KUKA KRL program: f1_Kuka_APT212T02S12.SRC

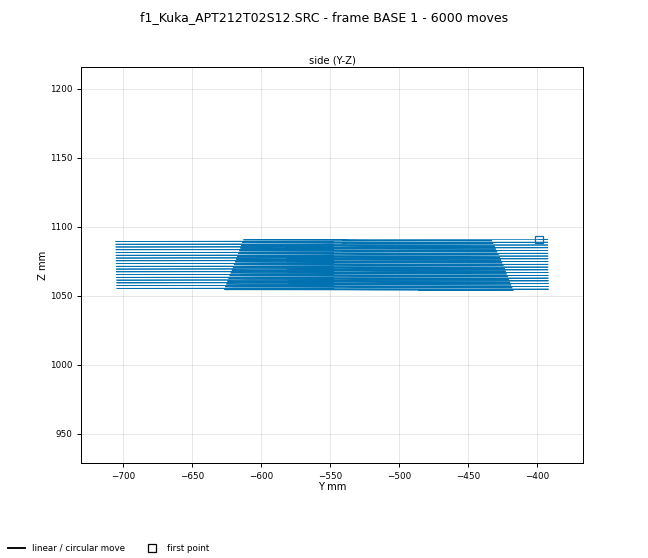
[picture p0: tool path of f1_Kuka_APT212T02S12.SRC in frame BASE 1, 6000 of 6001 moves have a stored position in this frame; points joined in program order, loops and branches not executed]
&ACCESS RVP
&REL 2
&PARAM TEMPLATE = C:\KRC\Roboter\Template\vorgabe
&PARAM EDITMASK = *
DEF f1_Kuka_APT212T02S12()


;FOLD INI;%{PE}%V3.2.0,%MKUKATPBASIS,%CINIT,%VCOMMON,%P
  ;FOLD BAS INI;%{E}%V3.2.0,%MKUKATPBASIS,%CINIT,%VINIT,%P
    GLOBAL INTERRUPT DECL 3 WHEN $STOPMESS==TRUE DO IR_STOPM ( )
    INTERRUPT ON 3
    BAS (#INITMOV,0 )
  ;ENDFOLD (BAS INI)
  ;FOLD USER INI;%{E}%V3.2.0,%MKUKATPUSER,%CINIT,%VINIT,%P
    ;Make your modifications here
  ;ENDFOLD (USER INI)
;ENDFOLD (INI)


;*** Make Null PTP Move
  PTP $pos_act

;*** Auto Load The Correct TOOL Data
  $tool=tool_data[2]

;*** Auto Load The Correct BASE Data
  $base=base_data[1]

  $ADVANCE = 5

;*** Restate Last Velocity
MMPM(30000.0)
SetRPM(8000)
LIN {X -0.086,Y -398.427,Z 1090.884,A 0.000,B 0.000,C 90.000,E1 15.190} C_DIS
LIN {X -0.036,Y -396.041,Z 1090.882,A 0.000,B 0.000,C 90.000,E1 14.773} C_DIS
LIN {X 0.107,Y -394.257,Z 1090.880,A 0.000,B 0.000,C 90.000,E1 14.356} C_DIS
LIN {X 0.038,Y -393.540,Z 1090.879,A 0.000,B 0.000,C 90.000,E1 14.189} C_DIS
LIN {X 0.038,Y -392.338,Z 1090.876,A 0.000,B 0.000,C 90.000,E1 13.647} C_DIS
LIN {X 0.042,Y -392.056,Z 1090.872,A 0.000,B 0.000,C 90.000,E1 12.939} C_DIS
LIN {X -0.016,Y -392.577,Z 1090.868,A 0.000,B 0.000,C 90.000,E1 12.243} C_DIS
LIN {X -0.109,Y -394.607,Z 1090.860,A 0.000,B 0.000,C 90.000,E1 10.838} C_DIS
LIN {X 0.062,Y -400.114,Z 1090.844,A 0.000,B 0.000,C 90.000,E1 7.992} C_DIS
LIN {X -0.050,Y -404.941,Z 1090.833,A 0.000,B 0.000,C 90.000,E1 5.910} C_DIS
LIN {X -0.108,Y -406.949,Z 1090.828,A 0.000,B 0.000,C 90.000,E1 5.049} C_DIS
LIN {X -0.130,Y -409.374,Z 1090.824,A 0.000,B 0.000,C 90.000,E1 4.359} C_DIS
LIN {X 0.208,Y -412.372,Z 1090.821,A 0.000,B 0.000,C 90.000,E1 3.784} C_DIS
LIN {X -0.071,Y -415.342,Z 1090.819,A 0.000,B 0.000,C 90.000,E1 3.498} C_DIS
LIN {X 0.069,Y -416.809,Z 1090.819,A 0.000,B 0.000,C 90.000,E1 3.326} C_DIS
LIN {X -0.093,Y -424.402,Z 1090.816,A 0.000,B 0.000,C 90.000,E1 2.808} C_DIS
LIN {X 0.127,Y -432.552,Z 1090.813,A 0.000,B 0.000,C 90.000,E1 2.236} C_DIS
LIN {X -0.175,Y -448.840,Z 1090.807,A 0.000,B 0.000,C 90.000,E1 1.203} C_DIS
LIN {X 0.179,Y -470.911,Z 1090.799,A 0.000,B 0.000,C 90.000,E1 359.771} C_DIS
LIN {X -0.123,Y -480.615,Z 1090.796,A 0.000,B 0.000,C 90.000,E1 359.198} C_DIS
LIN {X -0.067,Y -490.234,Z 1090.792,A 0.000,B 0.000,C 90.000,E1 358.568} C_DIS
LIN {X -0.141,Y -501.141,Z 1090.788,A 0.000,B 0.000,C 90.000,E1 357.822} C_DIS
LIN {X -0.002,Y -508.747,Z 1090.785,A 0.000,B 0.000,C 90.000,E1 357.249} C_DIS
LIN {X -0.176,Y -517.486,Z 1090.781,A 0.000,B 0.000,C 90.000,E1 356.560} C_DIS
LIN {X 0.062,Y -523.142,Z 1090.778,A 0.000,B 0.000,C 90.000,E1 356.045} C_DIS
LIN {X 0.124,Y -528.481,Z 1090.775,A 0.000,B 0.000,C 90.000,E1 355.527} C_DIS
LIN {X -0.033,Y -533.756,Z 1090.772,A 0.000,B 0.000,C 90.000,E1 355.008} C_DIS
LIN {X -0.006,Y -539.738,Z 1090.768,A 0.000,B 0.000,C 90.000,E1 354.318} C_DIS
LIN {X -0.098,Y -545.312,Z 1090.765,A 0.000,B 0.000,C 90.000,E1 353.628} C_DIS
LIN {X 0.005,Y -549.510,Z 1090.761,A 0.000,B 0.000,C 90.000,E1 353.053} C_DIS
LIN {X -0.044,Y -554.087,Z 1090.758,A 0.000,B 0.000,C 90.000,E1 352.356} C_DIS
LIN {X 0.122,Y -557.472,Z 1090.755,A 0.000,B 0.000,C 90.000,E1 351.781} C_DIS
LIN {X 0.146,Y -561.205,Z 1090.751,A 0.000,B 0.000,C 90.000,E1 351.084} C_DIS
LIN {X 0.207,Y -564.647,Z 1090.747,A 0.000,B 0.000,C 90.000,E1 350.387} C_DIS
LIN {X -0.087,Y -568.925,Z 1090.741,A 0.000,B 0.000,C 90.000,E1 349.454} C_DIS
LIN {X 0.100,Y -573.356,Z 1090.735,A 0.000,B 0.000,C 90.000,E1 348.342} C_DIS
LIN {X -0.002,Y -578.374,Z 1090.728,A 0.000,B 0.000,C 90.000,E1 346.992} C_DIS
LIN {X 0.202,Y -583.916,Z 1090.719,A 0.000,B 0.000,C 90.000,E1 345.353} C_DIS
LIN {X 0.003,Y -588.183,Z 1090.711,A 0.000,B 0.000,C 90.000,E1 344.031} C_DIS
LIN {X 0.030,Y -591.458,Z 1090.705,A 0.000,B 0.000,C 90.000,E1 342.960} C_DIS
LIN {X -0.029,Y -595.407,Z 1090.698,A 0.000,B 0.000,C 90.000,E1 341.638} C_DIS
LIN {X -0.187,Y -597.634,Z 1090.694,A 0.000,B 0.000,C 90.000,E1 340.859} C_DIS
LIN {X 0.046,Y -600.855,Z 1090.686,A 0.000,B 0.000,C 90.000,E1 339.518} C_DIS
LIN {X 0.066,Y -603.171,Z 1090.680,A 0.000,B 0.000,C 90.000,E1 338.465} C_DIS
LIN {X 0.124,Y -605.226,Z 1090.675,A 0.000,B 0.000,C 90.000,E1 337.411} C_DIS
LIN {X 0.209,Y -607.002,Z 1090.669,A 0.000,B 0.000,C 90.000,E1 336.357} C_DIS
LIN {X -0.245,Y -608.528,Z 1090.663,A 0.000,B 0.000,C 90.000,E1 335.357} C_DIS
LIN {X 0.127,Y -609.836,Z 1090.657,A 0.000,B 0.000,C 90.000,E1 334.280} C_DIS
LIN {X -0.030,Y -610.932,Z 1090.651,A 0.000,B 0.000,C 90.000,E1 333.256} C_DIS
LIN {X -0.211,Y -611.924,Z 1090.644,A 0.000,B 0.000,C 90.000,E1 331.975} C_DIS
LIN {X -0.023,Y -612.377,Z 1090.640,A 0.000,B 0.000,C 90.000,E1 331.179} C_DIS
LIN {X 0.141,Y -612.615,Z 1090.634,A 0.000,B 0.000,C 90.000,E1 330.127} C_DIS
LIN {X 0.342,Y -612.436,Z 1090.630,A 0.000,B 0.000,C 90.000,E1 329.331} C_DIS
LIN {X 0.017,Y -612.074,Z 1090.625,A 0.000,B 0.000,C 90.000,E1 328.584} C_DIS
LIN {X 0.210,Y -611.462,Z 1090.621,A 0.000,B 0.000,C 90.000,E1 327.788} C_DIS
LIN {X 0.156,Y -610.184,Z 1090.615,A 0.000,B 0.000,C 90.000,E1 326.755} C_DIS
LIN {X 0.088,Y -608.451,Z 1090.610,A 0.000,B 0.000,C 90.000,E1 325.722} C_DIS
LIN {X 0.262,Y -606.198,Z 1090.602,A 0.000,B 0.000,C 90.000,E1 324.402} C_DIS
LIN {X -0.099,Y -604.017,Z 1090.595,A 0.000,B 0.000,C 90.000,E1 323.130} C_DIS
LIN {X -0.134,Y -601.862,Z 1090.588,A 0.000,B 0.000,C 90.000,E1 321.823} C_DIS
LIN {X 0.148,Y -600.611,Z 1090.583,A 0.000,B 0.000,C 90.000,E1 321.009} C_DIS
LIN {X -0.208,Y -599.661,Z 1090.581,A 0.000,B 0.000,C 90.000,E1 320.517} C_DIS
LIN {X 0.031,Y -599.310,Z 1090.579,A 0.000,B 0.000,C 90.000,E1 320.231} C_DIS
LIN {X -0.190,Y -598.777,Z 1090.578,A 0.000,B 0.000,C 90.000,E1 319.989} C_DIS
LIN {X -0.177,Y -598.069,Z 1090.575,A 0.000,B 0.000,C 90.000,E1 319.461} C_DIS
LIN {X -0.169,Y -597.234,Z 1090.572,A 0.000,B 0.000,C 90.000,E1 318.933} C_DIS
LIN {X -0.168,Y -596.422,Z 1090.569,A 0.000,B 0.000,C 90.000,E1 318.405} C_DIS
LIN {X 0.214,Y -594.488,Z 1090.563,A 0.000,B 0.000,C 90.000,E1 317.310} C_DIS
LIN {X -0.269,Y -592.283,Z 1090.557,A 0.000,B 0.000,C 90.000,E1 316.296} C_DIS
LIN {X -0.134,Y -590.462,Z 1090.553,A 0.000,B 0.000,C 90.000,E1 315.486} C_DIS
LIN {X -0.170,Y -586.110,Z 1090.542,A 0.000,B 0.000,C 90.000,E1 313.623} C_DIS
LIN {X 0.151,Y -584.801,Z 1090.539,A 0.000,B 0.000,C 90.000,E1 313.056} C_DIS
LIN {X -0.129,Y -580.589,Z 1090.530,A 0.000,B 0.000,C 90.000,E1 311.472} C_DIS
LIN {X 0.142,Y -579.157,Z 1090.527,A 0.000,B 0.000,C 90.000,E1 310.906} C_DIS
LIN {X 0.176,Y -576.205,Z 1090.523,A 0.000,B 0.000,C 90.000,E1 310.092} C_DIS
LIN {X 0.037,Y -574.143,Z 1090.520,A 0.000,B 0.000,C 90.000,E1 309.564} C_DIS
LIN {X 0.155,Y -569.404,Z 1090.514,A 0.000,B 0.000,C 90.000,E1 308.463} C_DIS
LIN {X -0.031,Y -564.794,Z 1090.509,A 0.000,B 0.000,C 90.000,E1 307.523} C_DIS
LIN {X 0.190,Y -561.998,Z 1090.505,A 0.000,B 0.000,C 90.000,E1 306.950} C_DIS
LIN {X -0.178,Y -558.216,Z 1090.502,A 0.000,B 0.000,C 90.000,E1 306.297} C_DIS
LIN {X -0.008,Y -554.762,Z 1090.499,A 0.000,B 0.000,C 90.000,E1 305.724} C_DIS
LIN {X -0.057,Y -551.848,Z 1090.496,A 0.000,B 0.000,C 90.000,E1 305.311} C_DIS
LIN {X -0.064,Y -547.711,Z 1090.492,A 0.000,B 0.000,C 90.000,E1 304.612} C_DIS
LIN {X -0.016,Y -545.861,Z 1090.491,A 0.000,B 0.000,C 90.000,E1 304.326} C_DIS
LIN {X -0.244,Y -542.889,Z 1090.488,A 0.000,B 0.000,C 90.000,E1 303.785} C_DIS
LIN {X 0.261,Y -540.814,Z 1090.484,A 0.000,B 0.000,C 90.000,E1 303.166} C_DIS
LIN {X 0.155,Y -539.184,Z 1090.480,A 0.000,B 0.000,C 90.000,E1 302.467} C_DIS
LIN {X 0.179,Y -538.819,Z 1090.479,A 0.000,B 0.000,C 90.000,E1 302.133} C_DIS
LIN {X -0.101,Y -538.609,Z 1090.477,A 0.000,B 0.000,C 90.000,E1 301.878} C_DIS
LIN {X -0.096,Y -538.156,Z 1090.475,A 0.000,B 0.000,C 90.000,E1 301.592} C_DIS
LIN {X 0.085,Y -537.926,Z 1090.474,A 0.000,B 0.000,C 90.000,E1 301.288} C_DIS
LIN {X 0.150,Y -537.874,Z 1090.472,A 0.000,B 0.000,C 90.000,E1 301.003} C_DIS
LIN {X 0.147,Y -537.993,Z 1090.471,A 0.000,B 0.000,C 90.000,E1 300.718} C_DIS
LIN {X -0.132,Y -537.654,Z 1090.469,A 0.000,B 0.000,C 90.000,E1 300.463} C_DIS
LIN {X -0.308,Y -538.599,Z 1090.447,A 0.000,B 0.000,C 90.000,E1 296.488} C_DIS
LIN {X 0.034,Y -539.190,Z 1090.439,A 0.000,B 0.000,C 90.000,E1 295.027} C_DIS
LIN {X 0.166,Y -539.672,Z 1090.431,A 0.000,B 0.000,C 90.000,E1 293.590} C_DIS
LIN {X 0.033,Y -540.215,Z 1090.422,A 0.000,B 0.000,C 90.000,E1 291.897} C_DIS
LIN {X -0.030,Y -540.561,Z 1090.414,A 0.000,B 0.000,C 90.000,E1 290.482} C_DIS
LIN {X -0.275,Y -540.656,Z 1090.406,A 0.000,B 0.000,C 90.000,E1 289.087} C_DIS
LIN {X -0.227,Y -540.529,Z 1090.400,A 0.000,B 0.000,C 90.000,E1 287.946} C_DIS
LIN {X 0.039,Y -540.294,Z 1090.392,A 0.000,B 0.000,C 90.000,E1 286.496} C_DIS
LIN {X 0.203,Y -539.799,Z 1090.382,A 0.000,B 0.000,C 90.000,E1 284.773} C_DIS
LIN {X 0.153,Y -539.168,Z 1090.374,A 0.000,B 0.000,C 90.000,E1 283.355} C_DIS
LIN {X -0.027,Y -538.495,Z 1090.366,A 0.000,B 0.000,C 90.000,E1 281.951} C_DIS
LIN {X -0.218,Y -537.760,Z 1090.359,A 0.000,B 0.000,C 90.000,E1 280.546} C_DIS
LIN {X 0.010,Y -537.088,Z 1090.351,A 0.000,B 0.000,C 90.000,E1 279.095} C_DIS
LIN {X -0.268,Y -536.057,Z 1090.339,A 0.000,B 0.000,C 90.000,E1 277.125} C_DIS
LIN {X -0.103,Y -535.245,Z 1090.330,A 0.000,B 0.000,C 90.000,E1 275.391} C_DIS
LIN {X -0.045,Y -534.093,Z 1090.317,A 0.000,B 0.000,C 90.000,E1 273.094} C_DIS
LIN {X -0.069,Y -533.037,Z 1090.304,A 0.000,B 0.000,C 90.000,E1 270.802} C_DIS
LIN {X -0.101,Y -532.288,Z 1090.297,A 0.000,B 0.000,C 90.000,E1 269.370} C_DIS
LIN {X -0.147,Y -531.316,Z 1090.287,A 0.000,B 0.000,C 90.000,E1 267.650} C_DIS
LIN {X -0.200,Y -530.464,Z 1090.279,A 0.000,B 0.000,C 90.000,E1 266.216} C_DIS
LIN {X -0.238,Y -529.531,Z 1090.271,A 0.000,B 0.000,C 90.000,E1 264.780} C_DIS
LIN {X -0.226,Y -528.880,Z 1090.266,A 0.000,B 0.000,C 90.000,E1 263.913} C_DIS
LIN {X -0.279,Y -528.109,Z 1090.261,A 0.000,B 0.000,C 90.000,E1 263.053} C_DIS
LIN {X -0.216,Y -526.239,Z 1090.252,A 0.000,B 0.000,C 90.000,E1 261.310} C_DIS
LIN {X -0.164,Y -524.132,Z 1090.240,A 0.000,B 0.000,C 90.000,E1 259.275} C_DIS
LIN {X -0.103,Y -522.944,Z 1090.234,A 0.000,B 0.000,C 90.000,E1 258.105} C_DIS
LIN {X -0.056,Y -521.283,Z 1090.224,A 0.000,B 0.000,C 90.000,E1 256.353} C_DIS
LIN {X 0.190,Y -519.569,Z 1090.214,A 0.000,B 0.000,C 90.000,E1 254.574} C_DIS
LIN {X 0.023,Y -517.402,Z 1090.203,A 0.000,B 0.000,C 90.000,E1 252.543} C_DIS
LIN {X -0.050,Y -515.164,Z 1090.192,A 0.000,B 0.000,C 90.000,E1 250.496} C_DIS
LIN {X -0.208,Y -513.874,Z 1090.185,A 0.000,B 0.000,C 90.000,E1 249.337} C_DIS
LIN {X -0.076,Y -512.072,Z 1090.177,A 0.000,B 0.000,C 90.000,E1 247.847} C_DIS
LIN {X 0.027,Y -510.158,Z 1090.169,A 0.000,B 0.000,C 90.000,E1 246.357} C_DIS
LIN {X -0.016,Y -508.348,Z 1090.162,A 0.000,B 0.000,C 90.000,E1 245.177} C_DIS
LIN {X -0.023,Y -505.922,Z 1090.154,A 0.000,B 0.000,C 90.000,E1 243.691} C_DIS
LIN {X 0.004,Y -504.492,Z 1090.149,A 0.000,B 0.000,C 90.000,E1 242.794} C_DIS
LIN {X -0.062,Y -502.029,Z 1090.141,A 0.000,B 0.000,C 90.000,E1 241.307} C_DIS
LIN {X 0.101,Y -498.891,Z 1090.131,A 0.000,B 0.000,C 90.000,E1 239.488} C_DIS
LIN {X 0.130,Y -496.801,Z 1090.124,A 0.000,B 0.000,C 90.000,E1 238.280} C_DIS
LIN {X 0.122,Y -495.153,Z 1090.119,A 0.000,B 0.000,C 90.000,E1 237.375} C_DIS
LIN {X -0.205,Y -491.745,Z 1090.109,A 0.000,B 0.000,C 90.000,E1 235.595} C_DIS
LIN {X -0.177,Y -488.784,Z 1090.100,A 0.000,B 0.000,C 90.000,E1 234.069} C_DIS
LIN {X -0.146,Y -486.406,Z 1090.094,A 0.000,B 0.000,C 90.000,E1 232.844} C_DIS
LIN {X -0.025,Y -483.277,Z 1090.085,A 0.000,B 0.000,C 90.000,E1 231.295} C_DIS
LIN {X -0.080,Y -480.708,Z 1090.078,A 0.000,B 0.000,C 90.000,E1 230.070} C_DIS
LIN {X -0.329,Y -476.867,Z 1090.068,A 0.000,B 0.000,C 90.000,E1 228.243} C_DIS
LIN {X -0.151,Y -472.084,Z 1090.054,A 0.000,B 0.000,C 90.000,E1 225.729} C_DIS
LIN {X -0.208,Y -468.066,Z 1090.042,A 0.000,B 0.000,C 90.000,E1 223.542} C_DIS
LIN {X 0.172,Y -465.067,Z 1090.033,A 0.000,B 0.000,C 90.000,E1 221.919} C_DIS
LIN {X 0.233,Y -461.505,Z 1090.022,A 0.000,B 0.000,C 90.000,E1 220.011} C_DIS
LIN {X -0.115,Y -458.564,Z 1090.014,A 0.000,B 0.000,C 90.000,E1 218.463} C_DIS
LIN {X 0.208,Y -455.116,Z 1090.003,A 0.000,B 0.000,C 90.000,E1 216.503} C_DIS
LIN {X 0.195,Y -452.321,Z 1089.994,A 0.000,B 0.000,C 90.000,E1 214.898} C_DIS
LIN {X 0.046,Y -450.006,Z 1089.987,A 0.000,B 0.000,C 90.000,E1 213.627} C_DIS
LIN {X -0.015,Y -447.787,Z 1089.980,A 0.000,B 0.000,C 90.000,E1 212.339} C_DIS
LIN {X 0.019,Y -444.410,Z 1089.969,A 0.000,B 0.000,C 90.000,E1 210.384} C_DIS
LIN {X -0.036,Y -440.736,Z 1089.956,A 0.000,B 0.000,C 90.000,E1 208.103} C_DIS
LIN {X 0.101,Y -435.648,Z 1089.936,A 0.000,B 0.000,C 90.000,E1 204.463} C_DIS
LIN {X 0.037,Y -433.167,Z 1089.923,A 0.000,B 0.000,C 90.000,E1 202.153} C_DIS
LIN {X -0.118,Y -432.631,Z 1089.916,A 0.000,B 0.000,C 90.000,E1 200.844} C_DIS
LIN {X 0.148,Y -432.819,Z 1089.910,A 0.000,B 0.000,C 90.000,E1 199.812} C_DIS
LIN {X 0.191,Y -433.420,Z 1089.906,A 0.000,B 0.000,C 90.000,E1 199.141} C_DIS
LIN {X -0.081,Y -435.004,Z 1089.901,A 0.000,B 0.000,C 90.000,E1 198.181} C_DIS
LIN {X -0.025,Y -436.647,Z 1089.897,A 0.000,B 0.000,C 90.000,E1 197.511} C_DIS
LIN {X 0.159,Y -439.745,Z 1089.892,A 0.000,B 0.000,C 90.000,E1 196.496} C_DIS
LIN {X 0.112,Y -444.855,Z 1089.885,A 0.000,B 0.000,C 90.000,E1 195.190} C_DIS
LIN {X 0.164,Y -456.278,Z 1089.870,A 0.000,B 0.000,C 90.000,E1 192.591} C_DIS
LIN {X -0.058,Y -460.863,Z 1089.865,A 0.000,B 0.000,C 90.000,E1 191.658} C_DIS
LIN {X -0.140,Y -465.504,Z 1089.859,A 0.000,B 0.000,C 90.000,E1 190.715} C_DIS
LIN {X -0.075,Y -468.813,Z 1089.856,A 0.000,B 0.000,C 90.000,E1 190.074} C_DIS
LIN {X -0.194,Y -472.599,Z 1089.852,A 0.000,B 0.000,C 90.000,E1 189.321} C_DIS
LIN {X 0.098,Y -474.289,Z 1089.850,A 0.000,B 0.000,C 90.000,E1 188.973} C_DIS
LIN {X -0.103,Y -479.620,Z 1089.844,A 0.000,B 0.000,C 90.000,E1 187.936} C_DIS
LIN {X 0.069,Y -485.064,Z 1089.838,A 0.000,B 0.000,C 90.000,E1 186.834} C_DIS
LIN {X -0.236,Y -490.322,Z 1089.832,A 0.000,B 0.000,C 90.000,E1 185.796} C_DIS
LIN {X -0.134,Y -496.944,Z 1089.824,A 0.000,B 0.000,C 90.000,E1 184.416} C_DIS
LIN {X -0.233,Y -504.229,Z 1089.816,A 0.000,B 0.000,C 90.000,E1 182.922} C_DIS
LIN {X 0.197,Y -512.902,Z 1089.806,A 0.000,B 0.000,C 90.000,E1 181.088} C_DIS
LIN {X -0.155,Y -520.097,Z 1089.798,A 0.000,B 0.000,C 90.000,E1 179.656} C_DIS
LIN {X 0.156,Y -527.331,Z 1089.790,A 0.000,B 0.000,C 90.000,E1 178.165} C_DIS
LIN {X -0.198,Y -536.562,Z 1089.780,A 0.000,B 0.000,C 90.000,E1 176.331} C_DIS
LIN {X -0.084,Y -543.539,Z 1089.772,A 0.000,B 0.000,C 90.000,E1 174.894} C_DIS
LIN {X 0.255,Y -551.899,Z 1089.762,A 0.000,B 0.000,C 90.000,E1 173.166} C_DIS
LIN {X -0.260,Y -560.082,Z 1089.753,A 0.000,B 0.000,C 90.000,E1 171.546} C_DIS
LIN {X -0.131,Y -566.707,Z 1089.745,A 0.000,B 0.000,C 90.000,E1 170.151} C_DIS
LIN {X 0.114,Y -573.062,Z 1089.738,A 0.000,B 0.000,C 90.000,E1 168.757} C_DIS
LIN {X 0.254,Y -578.637,Z 1089.731,A 0.000,B 0.000,C 90.000,E1 167.521} C_DIS
LIN {X 0.119,Y -582.785,Z 1089.726,A 0.000,B 0.000,C 90.000,E1 166.589} C_DIS
LIN {X -0.254,Y -588.499,Z 1089.718,A 0.000,B 0.000,C 90.000,E1 165.283} C_DIS
LIN {X -0.221,Y -592.795,Z 1089.712,A 0.000,B 0.000,C 90.000,E1 164.212} C_DIS
LIN {X -0.129,Y -596.808,Z 1089.706,A 0.000,B 0.000,C 90.000,E1 163.142} C_DIS
LIN {X 0.194,Y -600.573,Z 1089.700,A 0.000,B 0.000,C 90.000,E1 162.054} C_DIS
LIN {X 0.295,Y -604.968,Z 1089.693,A 0.000,B 0.000,C 90.000,E1 160.732} C_DIS
LIN {X 0.098,Y -609.053,Z 1089.686,A 0.000,B 0.000,C 90.000,E1 159.444} C_DIS
LIN {X 0.014,Y -612.200,Z 1089.680,A 0.000,B 0.000,C 90.000,E1 158.411} C_DIS
LIN {X 0.229,Y -614.406,Z 1089.676,A 0.000,B 0.000,C 90.000,E1 157.614} C_DIS
LIN {X -0.169,Y -618.738,Z 1089.667,A 0.000,B 0.000,C 90.000,E1 156.102} C_DIS
LIN {X 0.096,Y -621.386,Z 1089.661,A 0.000,B 0.000,C 90.000,E1 155.049} C_DIS
LIN {X 0.097,Y -624.653,Z 1089.654,A 0.000,B 0.000,C 90.000,E1 153.768} C_DIS
LIN {X 0.141,Y -627.168,Z 1089.649,A 0.000,B 0.000,C 90.000,E1 152.743} C_DIS
LIN {X -0.293,Y -630.738,Z 1089.640,A 0.000,B 0.000,C 90.000,E1 151.257} C_DIS
LIN {X 0.157,Y -633.517,Z 1089.633,A 0.000,B 0.000,C 90.000,E1 149.950} C_DIS
LIN {X -0.074,Y -636.759,Z 1089.625,A 0.000,B 0.000,C 90.000,E1 148.456} C_DIS
LIN {X 0.306,Y -639.862,Z 1089.616,A 0.000,B 0.000,C 90.000,E1 146.914} C_DIS
LIN {X 0.155,Y -642.295,Z 1089.609,A 0.000,B 0.000,C 90.000,E1 145.674} C_DIS
LIN {X -0.072,Y -645.172,Z 1089.601,A 0.000,B 0.000,C 90.000,E1 144.196} C_DIS
LIN {X 0.145,Y -647.954,Z 1089.593,A 0.000,B 0.000,C 90.000,E1 142.683} C_DIS
LIN {X 0.419,Y -650.745,Z 1089.584,A 0.000,B 0.000,C 90.000,E1 141.170} C_DIS
LIN {X -0.270,Y -653.698,Z 1089.576,A 0.000,B 0.000,C 90.000,E1 139.747} C_DIS
LIN {X -0.054,Y -657.592,Z 1089.565,A 0.000,B 0.000,C 90.000,E1 137.757} C_DIS
LIN {X -0.206,Y -661.174,Z 1089.556,A 0.000,B 0.000,C 90.000,E1 136.053} C_DIS
LIN {X -0.310,Y -666.280,Z 1089.544,A 0.000,B 0.000,C 90.000,E1 133.866} C_DIS
LIN {X 0.183,Y -669.940,Z 1089.536,A 0.000,B 0.000,C 90.000,E1 132.366} C_DIS
LIN {X -0.117,Y -674.850,Z 1089.525,A 0.000,B 0.000,C 90.000,E1 130.458} C_DIS
LIN {X -0.209,Y -679.639,Z 1089.514,A 0.000,B 0.000,C 90.000,E1 128.543} C_DIS
LIN {X 0.175,Y -683.417,Z 1089.506,A 0.000,B 0.000,C 90.000,E1 127.076} C_DIS
LIN {X 0.186,Y -686.458,Z 1089.500,A 0.000,B 0.000,C 90.000,E1 125.884} C_DIS
LIN {X 0.054,Y -688.731,Z 1089.494,A 0.000,B 0.000,C 90.000,E1 124.945} C_DIS
LIN {X 0.358,Y -692.196,Z 1089.486,A 0.000,B 0.000,C 90.000,E1 123.499} C_DIS
LIN {X 0.123,Y -695.084,Z 1089.480,A 0.000,B 0.000,C 90.000,E1 122.339} C_DIS
LIN {X -0.075,Y -697.857,Z 1089.473,A 0.000,B 0.000,C 90.000,E1 121.180} C_DIS
LIN {X 0.089,Y -699.296,Z 1089.469,A 0.000,B 0.000,C 90.000,E1 120.463} C_DIS
LIN {X -0.067,Y -700.996,Z 1089.464,A 0.000,B 0.000,C 90.000,E1 119.539} C_DIS
LIN {X 0.136,Y -701.989,Z 1089.460,A 0.000,B 0.000,C 90.000,E1 118.821} C_DIS
LIN {X 0.350,Y -702.820,Z 1089.456,A 0.000,B 0.000,C 90.000,E1 118.103} C_DIS
LIN {X 0.192,Y -703.825,Z 1089.450,A 0.000,B 0.000,C 90.000,E1 116.950} C_DIS
LIN {X -0.296,Y -705.017,Z 1089.442,A 0.000,B 0.000,C 90.000,E1 115.591} C_DIS
LIN {X 0.279,Y -705.272,Z 1089.439,A 0.000,B 0.000,C 90.000,E1 115.079} C_DIS
LIN {X -0.081,Y -705.294,Z 1089.437,A 0.000,B 0.000,C 90.000,E1 114.643} C_DIS
LIN {X 0.204,Y -704.753,Z 1089.434,A 0.000,B 0.000,C 90.000,E1 114.155} C_DIS
LIN {X -0.153,Y -704.352,Z 1089.433,A 0.000,B 0.000,C 90.000,E1 113.951} C_DIS
LIN {X 0.132,Y -702.683,Z 1089.430,A 0.000,B 0.000,C 90.000,E1 113.462} C_DIS
LIN {X -0.234,Y -701.490,Z 1089.429,A 0.000,B 0.000,C 90.000,E1 113.259} C_DIS
LIN {X 0.033,Y -697.713,Z 1089.427,A 0.000,B 0.000,C 90.000,E1 112.770} C_DIS
LIN {X 0.163,Y -696.456,Z 1089.426,A 0.000,B 0.000,C 90.000,E1 112.642} C_DIS
LIN {X 0.291,Y -694.466,Z 1089.425,A 0.000,B 0.000,C 90.000,E1 112.514} C_DIS
LIN {X 0.169,Y -687.151,Z 1089.423,A 0.000,B 0.000,C 90.000,E1 112.206} C_DIS
LIN {X -0.051,Y -684.897,Z 1089.423,A 0.000,B 0.000,C 90.000,E1 112.153} C_DIS
LIN {X 0.024,Y -675.825,Z 1089.422,A 0.000,B 0.000,C 90.000,E1 112.025} C_DIS
LIN {X -0.028,Y -604.808,Z 1089.422,A 0.000,B 0.000,C 90.000,E1 112.025} C_DIS
LIN {X -0.164,Y -600.949,Z 1089.421,A 0.000,B 0.000,C 90.000,E1 111.844} C_DIS
LIN {X -0.082,Y -596.421,Z 1089.420,A 0.000,B 0.000,C 90.000,E1 111.535} C_DIS
LIN {X 0.109,Y -586.219,Z 1089.415,A 0.000,B 0.000,C 90.000,E1 110.684} C_DIS
LIN {X -0.207,Y -576.459,Z 1089.410,A 0.000,B 0.000,C 90.000,E1 109.885} C_DIS
LIN {X -0.103,Y -575.095,Z 1089.410,A 0.000,B 0.000,C 90.000,E1 109.758} C_DIS
LIN {X -0.227,Y -569.062,Z 1089.407,A 0.000,B 0.000,C 90.000,E1 109.322} C_DIS
LIN {X 0.087,Y -560.876,Z 1089.404,A 0.000,B 0.000,C 90.000,E1 108.779} C_DIS
LIN {X -0.023,Y -554.397,Z 1089.402,A 0.000,B 0.000,C 90.000,E1 108.417} C_DIS
LIN {X 0.181,Y -549.521,Z 1089.401,A 0.000,B 0.000,C 90.000,E1 108.055} C_DIS
LIN {X 0.056,Y -548.089,Z 1089.399,A 0.000,B 0.000,C 90.000,E1 107.873} C_DIS
LIN {X 0.013,Y -548.062,Z 1089.399,A 0.000,B 0.000,C 90.000,E1 107.873} C_DIS
LIN {X -0.276,Y -547.700,Z 1089.398,A 0.000,B 0.000,C 90.000,E1 107.583} C_DIS
LIN {X -0.075,Y -547.929,Z 1089.394,A 0.000,B 0.000,C 90.000,E1 106.858} C_DIS
LIN {X -0.169,Y -548.528,Z 1089.389,A 0.000,B 0.000,C 90.000,E1 106.024} C_DIS
LIN {X -0.239,Y -549.880,Z 1089.378,A 0.000,B 0.000,C 90.000,E1 104.064} C_DIS
LIN {X 0.122,Y -551.468,Z 1089.367,A 0.000,B 0.000,C 90.000,E1 102.063} C_DIS
LIN {X 0.166,Y -552.809,Z 1089.359,A 0.000,B 0.000,C 90.000,E1 100.658} C_DIS
LIN {X -0.254,Y -554.877,Z 1089.349,A 0.000,B 0.000,C 90.000,E1 98.746} C_DIS
LIN {X -0.253,Y -556.387,Z 1089.341,A 0.000,B 0.000,C 90.000,E1 97.352} C_DIS
LIN {X 0.122,Y -557.648,Z 1089.335,A 0.000,B 0.000,C 90.000,E1 96.201} C_DIS
LIN {X -0.036,Y -558.705,Z 1089.328,A 0.000,B 0.000,C 90.000,E1 95.106} C_DIS
LIN {X 0.247,Y -559.426,Z 1089.324,A 0.000,B 0.000,C 90.000,E1 94.245} C_DIS
LIN {X 0.190,Y -560.344,Z 1089.316,A 0.000,B 0.000,C 90.000,E1 92.865} C_DIS
LIN {X 0.019,Y -560.983,Z 1089.310,A 0.000,B 0.000,C 90.000,E1 91.776} C_DIS
LIN {X 0.037,Y -561.803,Z 1089.301,A 0.000,B 0.000,C 90.000,E1 90.115} C_DIS
LIN {X 0.074,Y -562.503,Z 1089.292,A 0.000,B 0.000,C 90.000,E1 88.453} C_DIS
LIN {X 0.033,Y -563.084,Z 1089.284,A 0.000,B 0.000,C 90.000,E1 87.078} C_DIS
LIN {X 0.038,Y -563.621,Z 1089.276,A 0.000,B 0.000,C 90.000,E1 85.698} C_DIS
LIN {X 0.058,Y -564.161,Z 1089.269,A 0.000,B 0.000,C 90.000,E1 84.318} C_DIS
LIN {X -0.166,Y -564.757,Z 1089.258,A 0.000,B 0.000,C 90.000,E1 82.413} C_DIS
LIN {X -0.072,Y -565.248,Z 1089.250,A 0.000,B 0.000,C 90.000,E1 81.027} C_DIS
LIN {X -0.106,Y -566.034,Z 1089.240,A 0.000,B 0.000,C 90.000,E1 79.106} C_DIS
LIN {X -0.179,Y -566.772,Z 1089.230,A 0.000,B 0.000,C 90.000,E1 77.465} C_DIS
LIN {X 0.242,Y -567.996,Z 1089.218,A 0.000,B 0.000,C 90.000,E1 75.227} C_DIS
LIN {X 0.073,Y -569.712,Z 1089.204,A 0.000,B 0.000,C 90.000,E1 72.779} C_DIS
LIN {X -0.017,Y -571.020,Z 1089.195,A 0.000,B 0.000,C 90.000,E1 71.148} C_DIS
LIN {X -0.086,Y -572.452,Z 1089.186,A 0.000,B 0.000,C 90.000,E1 69.518} C_DIS
LIN {X -0.283,Y -573.181,Z 1089.182,A 0.000,B 0.000,C 90.000,E1 68.720} C_DIS
LIN {X -0.070,Y -574.770,Z 1089.171,A 0.000,B 0.000,C 90.000,E1 66.794} C_DIS
LIN {X 0.199,Y -575.835,Z 1089.164,A 0.000,B 0.000,C 90.000,E1 65.409} C_DIS
LIN {X -0.182,Y -576.961,Z 1089.155,A 0.000,B 0.000,C 90.000,E1 63.819} C_DIS
LIN {X 0.231,Y -577.998,Z 1089.146,A 0.000,B 0.000,C 90.000,E1 62.153} C_DIS
LIN {X -0.216,Y -578.818,Z 1089.138,A 0.000,B 0.000,C 90.000,E1 60.845} C_DIS
LIN {X 0.139,Y -579.590,Z 1089.130,A 0.000,B 0.000,C 90.000,E1 59.459} C_DIS
LIN {X -0.144,Y -580.458,Z 1089.121,A 0.000,B 0.000,C 90.000,E1 57.867} C_DIS
LIN {X -0.126,Y -580.980,Z 1089.115,A 0.000,B 0.000,C 90.000,E1 56.786} C_DIS
LIN {X -0.090,Y -581.617,Z 1089.108,A 0.000,B 0.000,C 90.000,E1 55.435} C_DIS
LIN {X -0.188,Y -582.250,Z 1089.099,A 0.000,B 0.000,C 90.000,E1 53.829} C_DIS
LIN {X -0.005,Y -582.501,Z 1089.094,A 0.000,B 0.000,C 90.000,E1 53.004} C_DIS
LIN {X 0.240,Y -582.741,Z 1089.089,A 0.000,B 0.000,C 90.000,E1 51.904} C_DIS
LIN {X 0.021,Y -582.694,Z 1089.080,A 0.000,B 0.000,C 90.000,E1 50.312} C_DIS
LIN {X 0.198,Y -582.443,Z 1089.074,A 0.000,B 0.000,C 90.000,E1 49.218} C_DIS
LIN {X 0.267,Y -582.187,Z 1089.069,A 0.000,B 0.000,C 90.000,E1 48.405} C_DIS
LIN {X -0.085,Y -581.522,Z 1089.060,A 0.000,B 0.000,C 90.000,E1 46.824} C_DIS
LIN {X 0.089,Y -580.962,Z 1089.054,A 0.000,B 0.000,C 90.000,E1 45.729} C_DIS
LIN {X -0.163,Y -580.147,Z 1089.048,A 0.000,B 0.000,C 90.000,E1 44.676} C_DIS
LIN {X -0.155,Y -579.400,Z 1089.044,A 0.000,B 0.000,C 90.000,E1 43.866} C_DIS
LIN {X -0.012,Y -578.194,Z 1089.038,A 0.000,B 0.000,C 90.000,E1 42.771} C_DIS
LIN {X 0.111,Y -576.737,Z 1089.032,A 0.000,B 0.000,C 90.000,E1 41.676} C_DIS
LIN {X 0.120,Y -575.463,Z 1089.027,A 0.000,B 0.000,C 90.000,E1 40.862} C_DIS
LIN {X -0.174,Y -573.643,Z 1089.021,A 0.000,B 0.000,C 90.000,E1 39.806} C_DIS
LIN {X -0.360,Y -570.873,Z 1089.014,A 0.000,B 0.000,C 90.000,E1 38.463} C_DIS
LIN {X 0.041,Y -568.929,Z 1089.009,A 0.000,B 0.000,C 90.000,E1 37.604} C_DIS
LIN {X -0.033,Y -566.684,Z 1089.004,A 0.000,B 0.000,C 90.000,E1 36.790} C_DIS
LIN {X -0.015,Y -564.120,Z 1089.000,A 0.000,B 0.000,C 90.000,E1 35.964} C_DIS
LIN {X 0.098,Y -563.221,Z 1088.998,A 0.000,B 0.000,C 90.000,E1 35.678} C_DIS
LIN {X -0.276,Y -559.027,Z 1088.992,A 0.000,B 0.000,C 90.000,E1 34.612} C_DIS
LIN {X -0.328,Y -555.516,Z 1088.988,A 0.000,B 0.000,C 90.000,E1 33.785} C_DIS
LIN {X 0.042,Y -551.533,Z 1088.983,A 0.000,B 0.000,C 90.000,E1 32.911} C_DIS
LIN {X 0.069,Y -546.568,Z 1088.977,A 0.000,B 0.000,C 90.000,E1 31.926} C_DIS
LIN {X 0.198,Y -541.282,Z 1088.972,A 0.000,B 0.000,C 90.000,E1 30.924} C_DIS
LIN {X 0.117,Y -534.473,Z 1088.966,A 0.000,B 0.000,C 90.000,E1 29.795} C_DIS
LIN {X 0.124,Y -529.787,Z 1088.962,A 0.000,B 0.000,C 90.000,E1 29.077} C_DIS
LIN {X 0.243,Y -525.777,Z 1088.958,A 0.000,B 0.000,C 90.000,E1 28.487} C_DIS
LIN {X -0.217,Y -522.681,Z 1088.956,A 0.000,B 0.000,C 90.000,E1 28.103} C_DIS
LIN {X 0.049,Y -514.540,Z 1088.950,A 0.000,B 0.000,C 90.000,E1 27.052} C_DIS
LIN {X 0.141,Y -508.048,Z 1088.946,A 0.000,B 0.000,C 90.000,E1 26.309} C_DIS
LIN {X 0.231,Y -502.730,Z 1088.943,A 0.000,B 0.000,C 90.000,E1 25.720} C_DIS
LIN {X -0.019,Y -494.568,Z 1088.938,A 0.000,B 0.000,C 90.000,E1 24.899} C_DIS
LIN {X -0.042,Y -488.960,Z 1088.935,A 0.000,B 0.000,C 90.000,E1 24.335} C_DIS
LIN {X -0.107,Y -477.381,Z 1088.929,A 0.000,B 0.000,C 90.000,E1 23.259} C_DIS
LIN {X -0.054,Y -471.540,Z 1088.926,A 0.000,B 0.000,C 90.000,E1 22.717} C_DIS
LIN {X 0.000,Y -457.967,Z 1088.920,A 0.000,B 0.000,C 90.000,E1 21.535} C_DIS
LIN {X -0.172,Y -441.851,Z 1088.912,A 0.000,B 0.000,C 90.000,E1 20.120} C_DIS
LIN {X -0.132,Y -430.227,Z 1088.906,A 0.000,B 0.000,C 90.000,E1 19.014} C_DIS
LIN {X 0.092,Y -416.281,Z 1088.897,A 0.000,B 0.000,C 90.000,E1 17.511} C_DIS
LIN {X -0.045,Y -405.620,Z 1088.890,A 0.000,B 0.000,C 90.000,E1 16.260} C_DIS
LIN {X 0.133,Y -399.045,Z 1088.885,A 0.000,B 0.000,C 90.000,E1 15.371} C_DIS
LIN {X -0.048,Y -395.343,Z 1088.882,A 0.000,B 0.000,C 90.000,E1 14.773} C_DIS
LIN {X 0.131,Y -393.924,Z 1088.880,A 0.000,B 0.000,C 90.000,E1 14.356} C_DIS
LIN {X 0.061,Y -393.206,Z 1088.879,A 0.000,B 0.000,C 90.000,E1 14.189} C_DIS
LIN {X -0.091,Y -392.129,Z 1088.875,A 0.000,B 0.000,C 90.000,E1 13.592} C_DIS
LIN {X 0.057,Y -392.164,Z 1088.871,A 0.000,B 0.000,C 90.000,E1 12.771} C_DIS
LIN {X 0.064,Y -393.130,Z 1088.866,A 0.000,B 0.000,C 90.000,E1 11.883} C_DIS
LIN {X -0.156,Y -397.974,Z 1088.850,A 0.000,B 0.000,C 90.000,E1 9.086} C_DIS
LIN {X 0.004,Y -404.983,Z 1088.833,A 0.000,B 0.000,C 90.000,E1 5.910} C_DIS
LIN {X -0.038,Y -406.506,Z 1088.829,A 0.000,B 0.000,C 90.000,E1 5.220} C_DIS
LIN {X -0.070,Y -407.479,Z 1088.827,A 0.000,B 0.000,C 90.000,E1 4.878} C_DIS
LIN {X -0.078,Y -409.273,Z 1088.824,A 0.000,B 0.000,C 90.000,E1 4.359} C_DIS
LIN {X -0.166,Y -412.135,Z 1088.821,A 0.000,B 0.000,C 90.000,E1 3.841} C_DIS
LIN {X 0.037,Y -412.697,Z 1088.821,A 0.000,B 0.000,C 90.000,E1 3.726} C_DIS
LIN {X -0.051,Y -417.157,Z 1088.818,A 0.000,B 0.000,C 90.000,E1 3.269} C_DIS
LIN {X -0.126,Y -421.852,Z 1088.816,A 0.000,B 0.000,C 90.000,E1 2.922} C_DIS
LIN {X 0.056,Y -429.349,Z 1088.813,A 0.000,B 0.000,C 90.000,E1 2.407} C_DIS
LIN {X -0.176,Y -448.932,Z 1088.806,A 0.000,B 0.000,C 90.000,E1 1.146} C_DIS
LIN {X 0.000,Y -466.750,Z 1088.800,A 0.000,B 0.000,C 90.000,E1 360.000} C_DIS
LIN {X -0.227,Y -478.221,Z 1088.796,A 0.000,B 0.000,C 90.000,E1 359.312} C_DIS
LIN {X -0.180,Y -486.222,Z 1088.793,A 0.000,B 0.000,C 90.000,E1 358.797} C_DIS
LIN {X 0.154,Y -492.517,Z 1088.791,A 0.000,B 0.000,C 90.000,E1 358.339} C_DIS
LIN {X 0.031,Y -503.476,Z 1088.787,A 0.000,B 0.000,C 90.000,E1 357.593} C_DIS
LIN {X 0.092,Y -509.565,Z 1088.784,A 0.000,B 0.000,C 90.000,E1 357.135} C_DIS
LIN {X -0.066,Y -516.942,Z 1088.781,A 0.000,B 0.000,C 90.000,E1 356.560} C_DIS
LIN {X 0.174,Y -523.948,Z 1088.777,A 0.000,B 0.000,C 90.000,E1 355.927} C_DIS
LIN {X -0.222,Y -527.993,Z 1088.775,A 0.000,B 0.000,C 90.000,E1 355.584} C_DIS
LIN {X 0.168,Y -533.306,Z 1088.772,A 0.000,B 0.000,C 90.000,E1 355.008} C_DIS
LIN {X 0.275,Y -539.325,Z 1088.769,A 0.000,B 0.000,C 90.000,E1 354.318} C_DIS
LIN {X 0.178,Y -544.973,Z 1088.765,A 0.000,B 0.000,C 90.000,E1 353.628} C_DIS
LIN {X -0.108,Y -549.141,Z 1088.762,A 0.000,B 0.000,C 90.000,E1 353.109} C_DIS
LIN {X -0.160,Y -553.773,Z 1088.758,A 0.000,B 0.000,C 90.000,E1 352.413} C_DIS
LIN {X 0.004,Y -557.227,Z 1088.755,A 0.000,B 0.000,C 90.000,E1 351.837} C_DIS
LIN {X 0.027,Y -561.014,Z 1088.751,A 0.000,B 0.000,C 90.000,E1 351.141} C_DIS
LIN {X 0.086,Y -564.506,Z 1088.747,A 0.000,B 0.000,C 90.000,E1 350.443} C_DIS
LIN {X 0.175,Y -567.644,Z 1088.743,A 0.000,B 0.000,C 90.000,E1 349.746} C_DIS
LIN {X 0.156,Y -571.162,Z 1088.739,A 0.000,B 0.000,C 90.000,E1 348.926} C_DIS
LIN {X 0.057,Y -574.391,Z 1088.734,A 0.000,B 0.000,C 90.000,E1 348.117} C_DIS
LIN {X -0.251,Y -578.431,Z 1088.728,A 0.000,B 0.000,C 90.000,E1 347.061} C_DIS
LIN {X 0.088,Y -584.048,Z 1088.719,A 0.000,B 0.000,C 90.000,E1 345.408} C_DIS
LIN {X 0.138,Y -589.193,Z 1088.710,A 0.000,B 0.000,C 90.000,E1 343.795} C_DIS
LIN {X 0.178,Y -592.460,Z 1088.704,A 0.000,B 0.000,C 90.000,E1 342.725} C_DIS
LIN {X -0.127,Y -595.647,Z 1088.698,A 0.000,B 0.000,C 90.000,E1 341.692} C_DIS
LIN {X 0.181,Y -598.589,Z 1088.692,A 0.000,B 0.000,C 90.000,E1 340.604} C_DIS
LIN {X -0.124,Y -601.774,Z 1088.685,A 0.000,B 0.000,C 90.000,E1 339.316} C_DIS
LIN {X -0.305,Y -604.052,Z 1088.679,A 0.000,B 0.000,C 90.000,E1 338.284} C_DIS
LIN {X -0.239,Y -606.102,Z 1088.673,A 0.000,B 0.000,C 90.000,E1 337.230} C_DIS
LIN {X -0.198,Y -608.248,Z 1088.666,A 0.000,B 0.000,C 90.000,E1 335.921} C_DIS
LIN {X 0.172,Y -609.679,Z 1088.660,A 0.000,B 0.000,C 90.000,E1 334.845} C_DIS
LIN {X -0.021,Y -611.223,Z 1088.653,A 0.000,B 0.000,C 90.000,E1 333.563} C_DIS
LIN {X -0.157,Y -612.119,Z 1088.647,A 0.000,B 0.000,C 90.000,E1 332.538} C_DIS
LIN {X -0.286,Y -612.890,Z 1088.642,A 0.000,B 0.000,C 90.000,E1 331.513} C_DIS
LIN {X -0.085,Y -613.194,Z 1088.637,A 0.000,B 0.000,C 90.000,E1 330.717} C_DIS
LIN {X 0.123,Y -613.371,Z 1088.633,A 0.000,B 0.000,C 90.000,E1 329.921} C_DIS
LIN {X 0.020,Y -613.189,Z 1088.629,A 0.000,B 0.000,C 90.000,E1 329.154} C_DIS
LIN {X -0.022,Y -612.670,Z 1088.623,A 0.000,B 0.000,C 90.000,E1 328.122} C_DIS
LIN {X 0.173,Y -611.851,Z 1088.619,A 0.000,B 0.000,C 90.000,E1 327.327} C_DIS
LIN {X -0.161,Y -610.954,Z 1088.614,A 0.000,B 0.000,C 90.000,E1 326.580} C_DIS
LIN {X -0.163,Y -609.783,Z 1088.610,A 0.000,B 0.000,C 90.000,E1 325.801} C_DIS
LIN {X -0.243,Y -608.114,Z 1088.604,A 0.000,B 0.000,C 90.000,E1 324.769} C_DIS
LIN {X -0.307,Y -605.653,Z 1088.595,A 0.000,B 0.000,C 90.000,E1 323.210} C_DIS
LIN {X -0.015,Y -602.496,Z 1088.584,A 0.000,B 0.000,C 90.000,E1 321.090} C_DIS
LIN {X -0.062,Y -599.891,Z 1088.574,A 0.000,B 0.000,C 90.000,E1 319.256} C_DIS
LIN {X 0.366,Y -598.362,Z 1088.568,A 0.000,B 0.000,C 90.000,E1 318.162} C_DIS
LIN {X -0.065,Y -596.606,Z 1088.562,A 0.000,B 0.000,C 90.000,E1 317.148} C_DIS
LIN {X 0.321,Y -594.642,Z 1088.556,A 0.000,B 0.000,C 90.000,E1 316.053} C_DIS
LIN {X 0.063,Y -592.969,Z 1088.552,A 0.000,B 0.000,C 90.000,E1 315.283} C_DIS
LIN {X -0.213,Y -591.337,Z 1088.547,A 0.000,B 0.000,C 90.000,E1 314.514} C_DIS
LIN {X 0.151,Y -590.312,Z 1088.544,A 0.000,B 0.000,C 90.000,E1 313.947} C_DIS
LIN {X -0.051,Y -586.879,Z 1088.535,A 0.000,B 0.000,C 90.000,E1 312.366} C_DIS
LIN {X 0.061,Y -585.196,Z 1088.531,A 0.000,B 0.000,C 90.000,E1 311.553} C_DIS
LIN {X 0.279,Y -582.693,Z 1088.525,A 0.000,B 0.000,C 90.000,E1 310.458} C_DIS
LIN {X 0.009,Y -581.982,Z 1088.523,A 0.000,B 0.000,C 90.000,E1 310.216} C_DIS
LIN {X 0.237,Y -578.366,Z 1088.517,A 0.000,B 0.000,C 90.000,E1 309.116} C_DIS
LIN {X 0.061,Y -574.101,Z 1088.511,A 0.000,B 0.000,C 90.000,E1 308.051} C_DIS
LIN {X 0.182,Y -569.480,Z 1088.505,A 0.000,B 0.000,C 90.000,E1 306.950} C_DIS
LIN {X -0.015,Y -567.030,Z 1088.502,A 0.000,B 0.000,C 90.000,E1 306.423} C_DIS
LIN {X 0.104,Y -561.186,Z 1088.496,A 0.000,B 0.000,C 90.000,E1 305.311} C_DIS
LIN {X 0.178,Y -556.779,Z 1088.492,A 0.000,B 0.000,C 90.000,E1 304.612} C_DIS
LIN {X 0.141,Y -554.043,Z 1088.490,A 0.000,B 0.000,C 90.000,E1 304.199} C_DIS
LIN {X 0.023,Y -547.768,Z 1088.485,A 0.000,B 0.000,C 90.000,E1 303.372} C_DIS
LIN {X -0.104,Y -546.814,Z 1088.485,A 0.000,B 0.000,C 90.000,E1 303.245} C_DIS
LIN {X 0.067,Y -546.099,Z 1088.484,A 0.000,B 0.000,C 90.000,E1 303.086} C_DIS
LIN {X -0.190,Y -544.341,Z 1088.482,A 0.000,B 0.000,C 90.000,E1 302.832} C_DIS
LIN {X -0.033,Y -542.110,Z 1088.479,A 0.000,B 0.000,C 90.000,E1 302.260} C_DIS
LIN {X -0.299,Y -541.189,Z 1088.478,A 0.000,B 0.000,C 90.000,E1 302.005} C_DIS
LIN {X 0.042,Y -540.146,Z 1088.475,A 0.000,B 0.000,C 90.000,E1 301.544} C_DIS
LIN {X -0.085,Y -539.478,Z 1088.473,A 0.000,B 0.000,C 90.000,E1 301.131} C_DIS
LIN {X 0.332,Y -539.599,Z 1088.472,A 0.000,B 0.000,C 90.000,E1 300.924} C_DIS
LIN {X 0.058,Y -539.304,Z 1088.470,A 0.000,B 0.000,C 90.000,E1 300.669} C_DIS
LIN {X 0.059,Y -538.842,Z 1088.469,A 0.000,B 0.000,C 90.000,E1 300.384} C_DIS
LIN {X -0.061,Y -538.630,Z 1088.466,A 0.000,B 0.000,C 90.000,E1 299.922} C_DIS
LIN {X 0.133,Y -538.410,Z 1088.465,A 0.000,B 0.000,C 90.000,E1 299.617} C_DIS
LIN {X 0.173,Y -538.460,Z 1088.463,A 0.000,B 0.000,C 90.000,E1 299.333} C_DIS
LIN {X 0.099,Y -538.298,Z 1088.460,A 0.000,B 0.000,C 90.000,E1 298.771} C_DIS
LIN {X -0.065,Y -538.524,Z 1088.450,A 0.000,B 0.000,C 90.000,E1 297.078} C_DIS
LIN {X 0.247,Y -539.241,Z 1088.441,A 0.000,B 0.000,C 90.000,E1 295.335} C_DIS
LIN {X 0.105,Y -539.852,Z 1088.432,A 0.000,B 0.000,C 90.000,E1 293.643} C_DIS
LIN {X -0.030,Y -540.396,Z 1088.422,A 0.000,B 0.000,C 90.000,E1 291.950} C_DIS
LIN {X -0.055,Y -540.789,Z 1088.412,A 0.000,B 0.000,C 90.000,E1 290.248} C_DIS
LIN {X 0.171,Y -540.920,Z 1088.406,A 0.000,B 0.000,C 90.000,E1 289.087} C_DIS
LIN {X -0.292,Y -540.812,Z 1088.400,A 0.000,B 0.000,C 90.000,E1 288.000} C_DIS
LIN {X -0.025,Y -540.584,Z 1088.392,A 0.000,B 0.000,C 90.000,E1 286.551} C_DIS
LIN {X 0.142,Y -540.145,Z 1088.383,A 0.000,B 0.000,C 90.000,E1 284.828} C_DIS
LIN {X 0.164,Y -539.408,Z 1088.373,A 0.000,B 0.000,C 90.000,E1 283.119} C_DIS
LIN {X 0.056,Y -538.562,Z 1088.364,A 0.000,B 0.000,C 90.000,E1 281.422} C_DIS
LIN {X -0.101,Y -537.568,Z 1088.352,A 0.000,B 0.000,C 90.000,E1 279.443} C_DIS
LIN {X 0.126,Y -536.816,Z 1088.344,A 0.000,B 0.000,C 90.000,E1 277.992} C_DIS
LIN {X -0.172,Y -535.878,Z 1088.333,A 0.000,B 0.000,C 90.000,E1 276.024} C_DIS
LIN {X -0.121,Y -534.948,Z 1088.324,A 0.000,B 0.000,C 90.000,E1 274.302} C_DIS
LIN {X -0.077,Y -534.268,Z 1088.316,A 0.000,B 0.000,C 90.000,E1 272.865} C_DIS
LIN {X -0.087,Y -533.354,Z 1088.305,A 0.000,B 0.000,C 90.000,E1 270.859} C_DIS
LIN {X -0.114,Y -532.614,Z 1088.297,A 0.000,B 0.000,C 90.000,E1 269.427} C_DIS
LIN {X -0.153,Y -531.633,Z 1088.287,A 0.000,B 0.000,C 90.000,E1 267.707} C_DIS
LIN {X -0.182,Y -531.004,Z 1088.281,A 0.000,B 0.000,C 90.000,E1 266.560} C_DIS
LIN {X -0.208,Y -529.692,Z 1088.270,A 0.000,B 0.000,C 90.000,E1 264.546} C_DIS
LIN {X -0.263,Y -528.440,Z 1088.262,A 0.000,B 0.000,C 90.000,E1 263.109} C_DIS
LIN {X -0.270,Y -526.533,Z 1088.252,A 0.000,B 0.000,C 90.000,E1 261.376} C_DIS
LIN {X -0.167,Y -525.020,Z 1088.244,A 0.000,B 0.000,C 90.000,E1 259.916} C_DIS
LIN {X -0.180,Y -523.602,Z 1088.236,A 0.000,B 0.000,C 90.000,E1 258.465} C_DIS
LIN {X 0.000,Y -521.311,Z 1088.223,A 0.000,B 0.000,C 90.000,E1 256.117} C_DIS
LIN {X 0.254,Y -519.871,Z 1088.215,A 0.000,B 0.000,C 90.000,E1 254.629} C_DIS
LIN {X 0.100,Y -517.732,Z 1088.203,A 0.000,B 0.000,C 90.000,E1 252.598} C_DIS
LIN {X 0.039,Y -515.470,Z 1088.192,A 0.000,B 0.000,C 90.000,E1 250.550} C_DIS
LIN {X -0.110,Y -514.217,Z 1088.185,A 0.000,B 0.000,C 90.000,E1 249.390} C_DIS
LIN {X -0.042,Y -511.996,Z 1088.176,A 0.000,B 0.000,C 90.000,E1 247.614} C_DIS
LIN {X -0.058,Y -510.459,Z 1088.169,A 0.000,B 0.000,C 90.000,E1 246.433} C_DIS
LIN {X 0.111,Y -508.655,Z 1088.162,A 0.000,B 0.000,C 90.000,E1 245.229} C_DIS
LIN {X 0.286,Y -505.360,Z 1088.151,A 0.000,B 0.000,C 90.000,E1 243.127} C_DIS
LIN {X -0.148,Y -502.350,Z 1088.141,A 0.000,B 0.000,C 90.000,E1 241.385} C_DIS
LIN {X -0.122,Y -498.661,Z 1088.129,A 0.000,B 0.000,C 90.000,E1 239.282} C_DIS
LIN {X -0.094,Y -496.553,Z 1088.123,A 0.000,B 0.000,C 90.000,E1 238.074} C_DIS
LIN {X 0.024,Y -493.748,Z 1088.114,A 0.000,B 0.000,C 90.000,E1 236.548} C_DIS
LIN {X -0.030,Y -491.450,Z 1088.107,A 0.000,B 0.000,C 90.000,E1 235.341} C_DIS
LIN {X 0.109,Y -487.873,Z 1088.097,A 0.000,B 0.000,C 90.000,E1 233.497} C_DIS
LIN {X -0.220,Y -486.700,Z 1088.094,A 0.000,B 0.000,C 90.000,E1 232.924} C_DIS
LIN {X 0.102,Y -482.923,Z 1088.084,A 0.000,B 0.000,C 90.000,E1 231.045} C_DIS
LIN {X -0.220,Y -479.620,Z 1088.075,A 0.000,B 0.000,C 90.000,E1 229.542} C_DIS
LIN {X 0.072,Y -476.455,Z 1088.067,A 0.000,B 0.000,C 90.000,E1 227.957} C_DIS
LIN {X -0.207,Y -472.304,Z 1088.054,A 0.000,B 0.000,C 90.000,E1 225.810} C_DIS
LIN {X -0.258,Y -468.270,Z 1088.042,A 0.000,B 0.000,C 90.000,E1 223.623} C_DIS
LIN {X 0.061,Y -465.854,Z 1088.035,A 0.000,B 0.000,C 90.000,E1 222.324} C_DIS
LIN {X -0.204,Y -462.261,Z 1088.025,A 0.000,B 0.000,C 90.000,E1 220.458} C_DIS
LIN {X -0.150,Y -458.702,Z 1088.014,A 0.000,B 0.000,C 90.000,E1 218.543} C_DIS
LIN {X -0.187,Y -455.785,Z 1088.005,A 0.000,B 0.000,C 90.000,E1 216.950} C_DIS
LIN {X -0.200,Y -452.362,Z 1087.995,A 0.000,B 0.000,C 90.000,E1 215.025} C_DIS
LIN {X -0.110,Y -448.299,Z 1087.982,A 0.000,B 0.000,C 90.000,E1 212.752} C_DIS
LIN {X 0.004,Y -444.277,Z 1087.969,A 0.000,B 0.000,C 90.000,E1 210.463} C_DIS
LIN {X 0.160,Y -440.514,Z 1087.957,A 0.000,B 0.000,C 90.000,E1 208.153} C_DIS
LIN {X 0.016,Y -436.517,Z 1087.942,A 0.000,B 0.000,C 90.000,E1 205.540} C_DIS
LIN {X 0.097,Y -434.799,Z 1087.935,A 0.000,B 0.000,C 90.000,E1 204.207} C_DIS
LIN {X 0.005,Y -432.322,Z 1087.922,A 0.000,B 0.000,C 90.000,E1 201.897} C_DIS
LIN {X -0.137,Y -431.734,Z 1087.916,A 0.000,B 0.000,C 90.000,E1 200.918} C_DIS
LIN {X 0.122,Y -431.767,Z 1087.911,A 0.000,B 0.000,C 90.000,E1 199.885} C_DIS
LIN {X 0.159,Y -432.128,Z 1087.907,A 0.000,B 0.000,C 90.000,E1 199.214} C_DIS
LIN {X -0.026,Y -432.431,Z 1087.905,A 0.000,B 0.000,C 90.000,E1 198.906} C_DIS
LIN {X 0.240,Y -434.054,Z 1087.900,A 0.000,B 0.000,C 90.000,E1 197.873} C_DIS
LIN {X 0.157,Y -435.736,Z 1087.896,A 0.000,B 0.000,C 90.000,E1 197.221} C_DIS
LIN {X 0.090,Y -437.743,Z 1087.892,A 0.000,B 0.000,C 90.000,E1 196.567} C_DIS
LIN {X 0.131,Y -442.746,Z 1087.885,A 0.000,B 0.000,C 90.000,E1 195.245} C_DIS
LIN {X -0.064,Y -456.543,Z 1087.868,A 0.000,B 0.000,C 90.000,E1 192.187} C_DIS
LIN {X 0.028,Y -459.661,Z 1087.864,A 0.000,B 0.000,C 90.000,E1 191.535} C_DIS
LIN {X -0.006,Y -468.533,Z 1087.854,A 0.000,B 0.000,C 90.000,E1 189.792} C_DIS
LIN {X 0.037,Y -476.621,Z 1087.846,A 0.000,B 0.000,C 90.000,E1 188.219} C_DIS
LIN {X 0.098,Y -484.553,Z 1087.837,A 0.000,B 0.000,C 90.000,E1 186.663} C_DIS
LIN {X -0.053,Y -490.593,Z 1087.830,A 0.000,B 0.000,C 90.000,E1 185.454} C_DIS
LIN {X -0.114,Y -496.567,Z 1087.824,A 0.000,B 0.000,C 90.000,E1 184.245} C_DIS
LIN {X -0.216,Y -503.931,Z 1087.815,A 0.000,B 0.000,C 90.000,E1 182.751} C_DIS
LIN {X 0.209,Y -512.688,Z 1087.805,A 0.000,B 0.000,C 90.000,E1 180.917} C_DIS
LIN {X 0.086,Y -520.669,Z 1087.796,A 0.000,B 0.000,C 90.000,E1 179.312} C_DIS
LIN {X 0.162,Y -527.235,Z 1087.789,A 0.000,B 0.000,C 90.000,E1 177.993} C_DIS
LIN {X 0.074,Y -535.813,Z 1087.779,A 0.000,B 0.000,C 90.000,E1 176.274} C_DIS
LIN {X 0.178,Y -542.839,Z 1087.771,A 0.000,B 0.000,C 90.000,E1 174.837} C_DIS
LIN {X -0.077,Y -549.869,Z 1087.764,A 0.000,B 0.000,C 90.000,E1 173.451} C_DIS
LIN {X 0.096,Y -557.454,Z 1087.755,A 0.000,B 0.000,C 90.000,E1 171.894} C_DIS
LIN {X 0.024,Y -562.836,Z 1087.749,A 0.000,B 0.000,C 90.000,E1 170.792} C_DIS
LIN {X 0.027,Y -568.128,Z 1087.743,A 0.000,B 0.000,C 90.000,E1 169.690} C_DIS
LIN {X -0.033,Y -573.852,Z 1087.736,A 0.000,B 0.000,C 90.000,E1 168.465} C_DIS
LIN {X 0.228,Y -578.791,Z 1087.730,A 0.000,B 0.000,C 90.000,E1 167.353} C_DIS
LIN {X -0.014,Y -583.520,Z 1087.724,A 0.000,B 0.000,C 90.000,E1 166.297} C_DIS
LIN {X -0.056,Y -588.110,Z 1087.718,A 0.000,B 0.000,C 90.000,E1 165.227} C_DIS
LIN {X -0.030,Y -592.436,Z 1087.712,A 0.000,B 0.000,C 90.000,E1 164.157} C_DIS
LIN {X 0.055,Y -596.465,Z 1087.706,A 0.000,B 0.000,C 90.000,E1 163.087} C_DIS
LIN {X -0.199,Y -600.245,Z 1087.700,A 0.000,B 0.000,C 90.000,E1 162.054} C_DIS
LIN {X 0.176,Y -603.830,Z 1087.694,A 0.000,B 0.000,C 90.000,E1 160.967} C_DIS
LIN {X -0.248,Y -607.996,Z 1087.687,A 0.000,B 0.000,C 90.000,E1 159.699} C_DIS
LIN {X 0.169,Y -611.963,Z 1087.680,A 0.000,B 0.000,C 90.000,E1 158.358} C_DIS
LIN {X -0.225,Y -614.901,Z 1087.674,A 0.000,B 0.000,C 90.000,E1 157.358} C_DIS
LIN {X -0.030,Y -618.527,Z 1087.667,A 0.000,B 0.000,C 90.000,E1 156.049} C_DIS
LIN {X -0.074,Y -621.170,Z 1087.661,A 0.000,B 0.000,C 90.000,E1 155.025} C_DIS
LIN {X -0.343,Y -623.798,Z 1087.656,A 0.000,B 0.000,C 90.000,E1 154.024} C_DIS
LIN {X -0.300,Y -626.960,Z 1087.648,A 0.000,B 0.000,C 90.000,E1 152.743} C_DIS
LIN {X 0.091,Y -629.971,Z 1087.641,A 0.000,B 0.000,C 90.000,E1 151.435} C_DIS
LIN {X -0.326,Y -632.785,Z 1087.634,A 0.000,B 0.000,C 90.000,E1 150.205} C_DIS
LIN {X -0.028,Y -636.070,Z 1087.626,A 0.000,B 0.000,C 90.000,E1 148.663} C_DIS
LIN {X -0.198,Y -639.183,Z 1087.618,A 0.000,B 0.000,C 90.000,E1 147.168} C_DIS
LIN {X 0.135,Y -641.187,Z 1087.612,A 0.000,B 0.000,C 90.000,E1 146.135} C_DIS
LIN {X 0.011,Y -643.607,Z 1087.605,A 0.000,B 0.000,C 90.000,E1 144.895} C_DIS
LIN {X 0.293,Y -645.987,Z 1087.598,A 0.000,B 0.000,C 90.000,E1 143.623} C_DIS
LIN {X 0.131,Y -648.766,Z 1087.590,A 0.000,B 0.000,C 90.000,E1 142.145} C_DIS
LIN {X 0.219,Y -653.127,Z 1087.577,A 0.000,B 0.000,C 90.000,E1 139.908} C_DIS
LIN {X -0.022,Y -657.041,Z 1087.567,A 0.000,B 0.000,C 90.000,E1 137.957} C_DIS
LIN {X 0.234,Y -661.141,Z 1087.556,A 0.000,B 0.000,C 90.000,E1 135.972} C_DIS
LIN {X 0.137,Y -665.692,Z 1087.545,A 0.000,B 0.000,C 90.000,E1 134.028} C_DIS
LIN {X -0.318,Y -669.954,Z 1087.535,A 0.000,B 0.000,C 90.000,E1 132.366} C_DIS
LIN {X -0.109,Y -674.865,Z 1087.525,A 0.000,B 0.000,C 90.000,E1 130.415} C_DIS
LIN {X -0.314,Y -679.052,Z 1087.515,A 0.000,B 0.000,C 90.000,E1 128.749} C_DIS
LIN {X 0.210,Y -683.434,Z 1087.506,A 0.000,B 0.000,C 90.000,E1 127.030} C_DIS
LIN {X -0.327,Y -686.511,Z 1087.499,A 0.000,B 0.000,C 90.000,E1 125.884} C_DIS
LIN {X 0.105,Y -688.759,Z 1087.494,A 0.000,B 0.000,C 90.000,E1 124.898} C_DIS
LIN {X 0.203,Y -691.660,Z 1087.487,A 0.000,B 0.000,C 90.000,E1 123.706} C_DIS
LIN {X 0.193,Y -695.114,Z 1087.479,A 0.000,B 0.000,C 90.000,E1 122.291} C_DIS
LIN {X 0.003,Y -697.878,Z 1087.473,A 0.000,B 0.000,C 90.000,E1 121.131} C_DIS
LIN {X -0.087,Y -698.912,Z 1087.470,A 0.000,B 0.000,C 90.000,E1 120.669} C_DIS
LIN {X 0.023,Y -701.019,Z 1087.464,A 0.000,B 0.000,C 90.000,E1 119.489} C_DIS
LIN {X -0.109,Y -702.208,Z 1087.459,A 0.000,B 0.000,C 90.000,E1 118.565} C_DIS
LIN {X 0.109,Y -702.954,Z 1087.455,A 0.000,B 0.000,C 90.000,E1 117.847} C_DIS
LIN {X -0.391,Y -704.182,Z 1087.447,A 0.000,B 0.000,C 90.000,E1 116.488} C_DIS
LIN {X 0.103,Y -705.159,Z 1087.441,A 0.000,B 0.000,C 90.000,E1 115.283} C_DIS
LIN {X 0.035,Y -705.212,Z 1087.437,A 0.000,B 0.000,C 90.000,E1 114.591} C_DIS
LIN {X -0.033,Y -704.667,Z 1087.434,A 0.000,B 0.000,C 90.000,E1 114.131} C_DIS
LIN {X -0.034,Y -704.172,Z 1087.433,A 0.000,B 0.000,C 90.000,E1 113.898} C_DIS
LIN {X -0.114,Y -702.535,Z 1087.430,A 0.000,B 0.000,C 90.000,E1 113.439} C_DIS
LIN {X -0.254,Y -701.986,Z 1087.430,A 0.000,B 0.000,C 90.000,E1 113.334} C_DIS
LIN {X 0.289,Y -698.352,Z 1087.427,A 0.000,B 0.000,C 90.000,E1 112.823} C_DIS
LIN {X 0.151,Y -697.345,Z 1087.426,A 0.000,B 0.000,C 90.000,E1 112.717} C_DIS
LIN {X 0.280,Y -695.884,Z 1087.426,A 0.000,B 0.000,C 90.000,E1 112.589} C_DIS
LIN {X -0.233,Y -693.515,Z 1087.425,A 0.000,B 0.000,C 90.000,E1 112.514} C_DIS
LIN {X -0.110,Y -686.594,Z 1087.423,A 0.000,B 0.000,C 90.000,E1 112.206} C_DIS
LIN {X -0.238,Y -684.164,Z 1087.423,A 0.000,B 0.000,C 90.000,E1 112.153} C_DIS
LIN {X 0.008,Y -676.032,Z 1087.422,A 0.000,B 0.000,C 90.000,E1 112.025} C_DIS
LIN {X -0.040,Y -605.042,Z 1087.422,A 0.000,B 0.000,C 90.000,E1 112.025} C_DIS
LIN {X 0.100,Y -601.506,Z 1087.422,A 0.000,B 0.000,C 90.000,E1 111.844} C_DIS
LIN {X 0.165,Y -596.096,Z 1087.419,A 0.000,B 0.000,C 90.000,E1 111.482} C_DIS
LIN {X 0.272,Y -577.679,Z 1087.411,A 0.000,B 0.000,C 90.000,E1 109.939} C_DIS
LIN {X -0.261,Y -574.892,Z 1087.410,A 0.000,B 0.000,C 90.000,E1 109.758} C_DIS
LIN {X 0.076,Y -568.784,Z 1087.407,A 0.000,B 0.000,C 90.000,E1 109.268} C_DIS
LIN {X -0.159,Y -560.482,Z 1087.404,A 0.000,B 0.000,C 90.000,E1 108.779} C_DIS
LIN {X 0.255,Y -554.045,Z 1087.402,A 0.000,B 0.000,C 90.000,E1 108.362} C_DIS
LIN {X 0.320,Y -549.635,Z 1087.401,A 0.000,B 0.000,C 90.000,E1 108.055} C_DIS
LIN {X 0.039,Y -547.977,Z 1087.399,A 0.000,B 0.000,C 90.000,E1 107.873} C_DIS
LIN {X -0.002,Y -547.967,Z 1087.399,A 0.000,B 0.000,C 90.000,E1 107.873} C_DIS
LIN {X 0.128,Y -547.631,Z 1087.398,A 0.000,B 0.000,C 90.000,E1 107.583} C_DIS
LIN {X -0.057,Y -547.753,Z 1087.395,A 0.000,B 0.000,C 90.000,E1 107.040} C_DIS
LIN {X 0.092,Y -548.539,Z 1087.388,A 0.000,B 0.000,C 90.000,E1 105.898} C_DIS
LIN {X 0.015,Y -549.890,Z 1087.377,A 0.000,B 0.000,C 90.000,E1 103.939} C_DIS
LIN {X -0.170,Y -551.763,Z 1087.365,A 0.000,B 0.000,C 90.000,E1 101.715} C_DIS
LIN {X -0.240,Y -552.834,Z 1087.359,A 0.000,B 0.000,C 90.000,E1 100.602} C_DIS
LIN {X -0.149,Y -554.627,Z 1087.349,A 0.000,B 0.000,C 90.000,E1 98.916} C_DIS
LIN {X -0.230,Y -556.145,Z 1087.342,A 0.000,B 0.000,C 90.000,E1 97.530} C_DIS
LIN {X -0.278,Y -557.722,Z 1087.334,A 0.000,B 0.000,C 90.000,E1 96.144} C_DIS
LIN {X 0.121,Y -558.754,Z 1087.328,A 0.000,B 0.000,C 90.000,E1 94.992} C_DIS
LIN {X -0.028,Y -559.673,Z 1087.322,A 0.000,B 0.000,C 90.000,E1 93.898} C_DIS
LIN {X -0.026,Y -560.699,Z 1087.313,A 0.000,B 0.000,C 90.000,E1 92.236} C_DIS
LIN {X -0.190,Y -561.254,Z 1087.306,A 0.000,B 0.000,C 90.000,E1 91.146} C_DIS
LIN {X 0.201,Y -561.801,Z 1087.300,A 0.000,B 0.000,C 90.000,E1 90.000} C_DIS
LIN {X 0.236,Y -562.484,Z 1087.291,A 0.000,B 0.000,C 90.000,E1 88.339} C_DIS
LIN {X -0.237,Y -563.166,Z 1087.282,A 0.000,B 0.000,C 90.000,E1 86.731} C_DIS
LIN {X -0.267,Y -563.676,Z 1087.274,A 0.000,B 0.000,C 90.000,E1 85.355} C_DIS
LIN {X 0.215,Y -564.089,Z 1087.268,A 0.000,B 0.000,C 90.000,E1 84.204} C_DIS
LIN {X -0.015,Y -564.703,Z 1087.257,A 0.000,B 0.000,C 90.000,E1 82.299} C_DIS
LIN {X 0.162,Y -565.188,Z 1087.250,A 0.000,B 0.000,C 90.000,E1 80.905} C_DIS
LIN {X 0.033,Y -565.992,Z 1087.239,A 0.000,B 0.000,C 90.000,E1 78.993} C_DIS
LIN {X 0.123,Y -566.867,Z 1087.228,A 0.000,B 0.000,C 90.000,E1 77.061} C_DIS
LIN {X -0.244,Y -568.316,Z 1087.214,A 0.000,B 0.000,C 90.000,E1 74.629} C_DIS
LIN {X -0.026,Y -569.934,Z 1087.202,A 0.000,B 0.000,C 90.000,E1 72.417} C_DIS
LIN {X 0.050,Y -571.507,Z 1087.192,A 0.000,B 0.000,C 90.000,E1 70.496} C_DIS
LIN {X 0.179,Y -572.958,Z 1087.183,A 0.000,B 0.000,C 90.000,E1 68.847} C_DIS
LIN {X 0.222,Y -574.753,Z 1087.171,A 0.000,B 0.000,C 90.000,E1 66.666} C_DIS
LIN {X 0.097,Y -575.992,Z 1087.161,A 0.000,B 0.000,C 90.000,E1 65.049} C_DIS
LIN {X -0.036,Y -577.068,Z 1087.152,A 0.000,B 0.000,C 90.000,E1 63.435} C_DIS
LIN {X -0.132,Y -578.118,Z 1087.143,A 0.000,B 0.000,C 90.000,E1 61.820} C_DIS
LIN {X -0.218,Y -579.053,Z 1087.134,A 0.000,B 0.000,C 90.000,E1 60.205} C_DIS
LIN {X -0.219,Y -579.625,Z 1087.128,A 0.000,B 0.000,C 90.000,E1 59.125} C_DIS
LIN {X 0.289,Y -580.209,Z 1087.122,A 0.000,B 0.000,C 90.000,E1 57.995} C_DIS
LIN {X -0.333,Y -580.874,Z 1087.115,A 0.000,B 0.000,C 90.000,E1 56.707} C_DIS
LIN {X 0.184,Y -581.475,Z 1087.107,A 0.000,B 0.000,C 90.000,E1 55.308} C_DIS
LIN {X 0.253,Y -582.221,Z 1087.097,A 0.000,B 0.000,C 90.000,E1 53.417} C_DIS
LIN {X -0.143,Y -582.474,Z 1087.089,A 0.000,B 0.000,C 90.000,E1 52.110} C_DIS
LIN {X 0.212,Y -582.512,Z 1087.086,A 0.000,B 0.000,C 90.000,E1 51.537} C_DIS
LIN {X 0.186,Y -582.402,Z 1087.079,A 0.000,B 0.000,C 90.000,E1 50.194} C_DIS
LIN {X -0.012,Y -582.148,Z 1087.073,A 0.000,B 0.000,C 90.000,E1 49.138} C_DIS
LIN {X -0.214,Y -581.761,Z 1087.067,A 0.000,B 0.000,C 90.000,E1 48.081} C_DIS
LIN {X 0.121,Y -581.218,Z 1087.060,A 0.000,B 0.000,C 90.000,E1 46.701} C_DIS
LIN {X -0.132,Y -580.584,Z 1087.054,A 0.000,B 0.000,C 90.000,E1 45.648} C_DIS
LIN {X -0.119,Y -579.980,Z 1087.049,A 0.000,B 0.000,C 90.000,E1 44.838} C_DIS
LIN {X -0.111,Y -579.232,Z 1087.045,A 0.000,B 0.000,C 90.000,E1 44.028} C_DIS
LIN {X -0.117,Y -578.328,Z 1087.040,A 0.000,B 0.000,C 90.000,E1 43.218} C_DIS
LIN {X -0.249,Y -577.701,Z 1087.037,A 0.000,B 0.000,C 90.000,E1 42.690} C_DIS
LIN {X 0.013,Y -575.801,Z 1087.030,A 0.000,B 0.000,C 90.000,E1 41.310} C_DIS
LIN {X 0.016,Y -574.484,Z 1087.025,A 0.000,B 0.000,C 90.000,E1 40.496} C_DIS
LIN {X 0.074,Y -572.431,Z 1087.019,A 0.000,B 0.000,C 90.000,E1 39.402} C_DIS
LIN {X 0.171,Y -570.135,Z 1087.013,A 0.000,B 0.000,C 90.000,E1 38.302} C_DIS
LIN {X -0.367,Y -568.869,Z 1087.010,A 0.000,B 0.000,C 90.000,E1 37.810} C_DIS
LIN {X 0.133,Y -565.794,Z 1087.004,A 0.000,B 0.000,C 90.000,E1 36.664} C_DIS
LIN {X -0.091,Y -564.066,Z 1087.001,A 0.000,B 0.000,C 90.000,E1 36.137} C_DIS
LIN {X -0.203,Y -562.173,Z 1086.998,A 0.000,B 0.000,C 90.000,E1 35.598} C_DIS
LIN {X -0.131,Y -557.903,Z 1086.992,A 0.000,B 0.000,C 90.000,E1 34.485} C_DIS
LIN {X -0.079,Y -554.924,Z 1086.988,A 0.000,B 0.000,C 90.000,E1 33.785} C_DIS
LIN {X -0.058,Y -551.630,Z 1086.984,A 0.000,B 0.000,C 90.000,E1 33.086} C_DIS
LIN {X 0.137,Y -546.690,Z 1086.978,A 0.000,B 0.000,C 90.000,E1 32.084} C_DIS
LIN {X 0.071,Y -542.918,Z 1086.974,A 0.000,B 0.000,C 90.000,E1 31.386} C_DIS
LIN {X 0.286,Y -539.808,Z 1086.971,A 0.000,B 0.000,C 90.000,E1 30.797} C_DIS
LIN {X 0.327,Y -533.853,Z 1086.966,A 0.000,B 0.000,C 90.000,E1 29.795} C_DIS
LIN {X -0.135,Y -529.114,Z 1086.962,A 0.000,B 0.000,C 90.000,E1 29.127} C_DIS
LIN {X -0.022,Y -525.059,Z 1086.959,A 0.000,B 0.000,C 90.000,E1 28.537} C_DIS
LIN {X -0.027,Y -521.912,Z 1086.956,A 0.000,B 0.000,C 90.000,E1 28.103} C_DIS
LIN {X -0.005,Y -513.728,Z 1086.950,A 0.000,B 0.000,C 90.000,E1 27.078} C_DIS
LIN {X -0.134,Y -507.218,Z 1086.946,A 0.000,B 0.000,C 90.000,E1 26.360} C_DIS
LIN {X -0.169,Y -501.980,Z 1086.943,A 0.000,B 0.000,C 90.000,E1 25.796} C_DIS
LIN {X 0.148,Y -492.458,Z 1086.938,A 0.000,B 0.000,C 90.000,E1 24.771} C_DIS
LIN {X 0.223,Y -486.734,Z 1086.935,A 0.000,B 0.000,C 90.000,E1 24.207} C_DIS
LIN {X -0.059,Y -478.506,Z 1086.930,A 0.000,B 0.000,C 90.000,E1 23.462} C_DIS
LIN {X 0.192,Y -471.342,Z 1086.927,A 0.000,B 0.000,C 90.000,E1 22.770} C_DIS
LIN {X -0.131,Y -458.068,Z 1086.920,A 0.000,B 0.000,C 90.000,E1 21.663} C_DIS
LIN {X -0.104,Y -446.146,Z 1086.914,A 0.000,B 0.000,C 90.000,E1 20.610} C_DIS
LIN {X 0.155,Y -431.532,Z 1086.907,A 0.000,B 0.000,C 90.000,E1 19.214} C_DIS
LIN {X -0.197,Y -416.028,Z 1086.898,A 0.000,B 0.000,C 90.000,E1 17.638} C_DIS
LIN {X 0.180,Y -405.368,Z 1086.891,A 0.000,B 0.000,C 90.000,E1 16.315} C_DIS
LIN {X 0.137,Y -399.049,Z 1086.886,A 0.000,B 0.000,C 90.000,E1 15.481} C_DIS
LIN {X 0.013,Y -397.057,Z 1086.884,A 0.000,B 0.000,C 90.000,E1 15.190} C_DIS
LIN {X -0.128,Y -395.332,Z 1086.883,A 0.000,B 0.000,C 90.000,E1 14.898} C_DIS
LIN {X -0.095,Y -394.560,Z 1086.882,A 0.000,B 0.000,C 90.000,E1 14.717} C_DIS
LIN {X -0.009,Y -392.788,Z 1086.879,A 0.000,B 0.000,C 90.000,E1 14.175} C_DIS
LIN {X 0.093,Y -392.039,Z 1086.875,A 0.000,B 0.000,C 90.000,E1 13.536} C_DIS
LIN {X 0.066,Y -392.088,Z 1086.872,A 0.000,B 0.000,C 90.000,E1 13.008} C_DIS
LIN {X 0.010,Y -393.200,Z 1086.866,A 0.000,B 0.000,C 90.000,E1 11.951} C_DIS
LIN {X -0.195,Y -397.975,Z 1086.851,A 0.000,B 0.000,C 90.000,E1 9.151} C_DIS
LIN {X 0.026,Y -404.897,Z 1086.833,A 0.000,B 0.000,C 90.000,E1 5.967} C_DIS
LIN {X -0.051,Y -407.287,Z 1086.827,A 0.000,B 0.000,C 90.000,E1 4.935} C_DIS
LIN {X -0.018,Y -408.967,Z 1086.825,A 0.000,B 0.000,C 90.000,E1 4.416} C_DIS
LIN {X -0.127,Y -410.731,Z 1086.823,A 0.000,B 0.000,C 90.000,E1 4.069} C_DIS
LIN {X -0.142,Y -412.634,Z 1086.821,A 0.000,B 0.000,C 90.000,E1 3.726} C_DIS
LIN {X 0.170,Y -416.400,Z 1086.818,A 0.000,B 0.000,C 90.000,E1 3.269} C_DIS
LIN {X -0.099,Y -421.792,Z 1086.816,A 0.000,B 0.000,C 90.000,E1 2.865} C_DIS
LIN {X 0.054,Y -429.400,Z 1086.813,A 0.000,B 0.000,C 90.000,E1 2.350} C_DIS
LIN {X 0.219,Y -447.385,Z 1086.807,A 0.000,B 0.000,C 90.000,E1 1.146} C_DIS
LIN {X -0.146,Y -465.332,Z 1086.800,A 0.000,B 0.000,C 90.000,E1 0.057} C_DIS
LIN {X 0.138,Y -475.821,Z 1086.797,A 0.000,B 0.000,C 90.000,E1 359.370} C_DIS
LIN {X -0.095,Y -485.360,Z 1086.793,A 0.000,B 0.000,C 90.000,E1 358.797} C_DIS
LIN {X 0.239,Y -491.710,Z 1086.791,A 0.000,B 0.000,C 90.000,E1 358.339} C_DIS
LIN {X 0.104,Y -502.769,Z 1086.787,A 0.000,B 0.000,C 90.000,E1 357.593} C_DIS
LIN {X 0.166,Y -510.336,Z 1086.784,A 0.000,B 0.000,C 90.000,E1 357.020} C_DIS
LIN {X 0.080,Y -516.344,Z 1086.781,A 0.000,B 0.000,C 90.000,E1 356.560} C_DIS
LIN {X -0.244,Y -523.466,Z 1086.778,A 0.000,B 0.000,C 90.000,E1 355.988} C_DIS
LIN {X 0.053,Y -527.398,Z 1086.776,A 0.000,B 0.000,C 90.000,E1 355.584} C_DIS
LIN {X -0.158,Y -532.837,Z 1086.773,A 0.000,B 0.000,C 90.000,E1 355.065} C_DIS
LIN {X -0.082,Y -538.998,Z 1086.769,A 0.000,B 0.000,C 90.000,E1 354.375} C_DIS
LIN {X -0.221,Y -544.716,Z 1086.765,A 0.000,B 0.000,C 90.000,E1 353.685} C_DIS
LIN {X -0.123,Y -549.082,Z 1086.762,A 0.000,B 0.000,C 90.000,E1 353.109} C_DIS
LIN {X -0.176,Y -553.748,Z 1086.758,A 0.000,B 0.000,C 90.000,E1 352.413} C_DIS
LIN {X -0.013,Y -557.237,Z 1086.755,A 0.000,B 0.000,C 90.000,E1 351.837} C_DIS
LIN {X 0.010,Y -561.056,Z 1086.751,A 0.000,B 0.000,C 90.000,E1 351.141} C_DIS
LIN {X 0.069,Y -564.583,Z 1086.747,A 0.000,B 0.000,C 90.000,E1 350.443} C_DIS
LIN {X -0.255,Y -567.173,Z 1086.744,A 0.000,B 0.000,C 90.000,E1 349.926} C_DIS
LIN {X -0.042,Y -570.150,Z 1086.740,A 0.000,B 0.000,C 90.000,E1 349.218} C_DIS
LIN {X -0.151,Y -573.502,Z 1086.736,A 0.000,B 0.000,C 90.000,E1 348.409} C_DIS
LIN {X 0.092,Y -577.620,Z 1086.729,A 0.000,B 0.000,C 90.000,E1 347.297} C_DIS
LIN {X 0.305,Y -580.536,Z 1086.725,A 0.000,B 0.000,C 90.000,E1 346.464} C_DIS
LIN {X -0.251,Y -585.196,Z 1086.718,A 0.000,B 0.000,C 90.000,E1 345.172} C_DIS
LIN {X -0.179,Y -590.343,Z 1086.709,A 0.000,B 0.000,C 90.000,E1 343.559} C_DIS
LIN {X 0.308,Y -594.396,Z 1086.701,A 0.000,B 0.000,C 90.000,E1 342.181} C_DIS
LIN {X 0.143,Y -596.769,Z 1086.697,A 0.000,B 0.000,C 90.000,E1 341.402} C_DIS
LIN {X 0.195,Y -598.941,Z 1086.692,A 0.000,B 0.000,C 90.000,E1 340.604} C_DIS
LIN {X -0.103,Y -602.194,Z 1086.685,A 0.000,B 0.000,C 90.000,E1 339.316} C_DIS
LIN {X -0.280,Y -604.508,Z 1086.679,A 0.000,B 0.000,C 90.000,E1 338.284} C_DIS
LIN {X -0.206,Y -606.563,Z 1086.673,A 0.000,B 0.000,C 90.000,E1 337.230} C_DIS
LIN {X -0.108,Y -608.320,Z 1086.668,A 0.000,B 0.000,C 90.000,E1 336.177} C_DIS
LIN {X 0.219,Y -610.207,Z 1086.660,A 0.000,B 0.000,C 90.000,E1 334.845} C_DIS
LIN {X 0.035,Y -611.768,Z 1086.653,A 0.000,B 0.000,C 90.000,E1 333.563} C_DIS
LIN {X -0.061,Y -612.528,Z 1086.649,A 0.000,B 0.000,C 90.000,E1 332.794} C_DIS
LIN {X -0.213,Y -613.523,Z 1086.642,A 0.000,B 0.000,C 90.000,E1 331.513} C_DIS
LIN {X -0.006,Y -613.880,Z 1086.637,A 0.000,B 0.000,C 90.000,E1 330.717} C_DIS
LIN {X 0.179,Y -614.108,Z 1086.632,A 0.000,B 0.000,C 90.000,E1 329.665} C_DIS
LIN {X -0.132,Y -613.923,Z 1086.627,A 0.000,B 0.000,C 90.000,E1 328.918} C_DIS
LIN {X 0.044,Y -613.394,Z 1086.622,A 0.000,B 0.000,C 90.000,E1 327.867} C_DIS
LIN {X -0.037,Y -612.060,Z 1086.614,A 0.000,B 0.000,C 90.000,E1 326.580} C_DIS
LIN {X -0.029,Y -610.996,Z 1086.610,A 0.000,B 0.000,C 90.000,E1 325.801} C_DIS
LIN {X 0.188,Y -609.111,Z 1086.603,A 0.000,B 0.000,C 90.000,E1 324.482} C_DIS
LIN {X 0.144,Y -606.801,Z 1086.594,A 0.000,B 0.000,C 90.000,E1 322.924} C_DIS
LIN {X -0.055,Y -604.652,Z 1086.585,A 0.000,B 0.000,C 90.000,E1 321.376} C_DIS
LIN {X -0.041,Y -602.300,Z 1086.575,A 0.000,B 0.000,C 90.000,E1 319.542} C_DIS
LIN {X -0.185,Y -600.615,Z 1086.568,A 0.000,B 0.000,C 90.000,E1 318.243} C_DIS
LIN {X -0.374,Y -599.489,Z 1086.564,A 0.000,B 0.000,C 90.000,E1 317.472} C_DIS
LIN {X -0.163,Y -597.238,Z 1086.556,A 0.000,B 0.000,C 90.000,E1 316.134} C_DIS
LIN {X -0.196,Y -595.352,Z 1086.550,A 0.000,B 0.000,C 90.000,E1 315.081} C_DIS
LIN {X -0.027,Y -593.892,Z 1086.546,A 0.000,B 0.000,C 90.000,E1 314.271} C_DIS
LIN {X 0.354,Y -593.001,Z 1086.543,A 0.000,B 0.000,C 90.000,E1 313.704} C_DIS
LIN {X -0.189,Y -590.134,Z 1086.534,A 0.000,B 0.000,C 90.000,E1 312.162} C_DIS
LIN {X -0.149,Y -587.559,Z 1086.527,A 0.000,B 0.000,C 90.000,E1 310.825} C_DIS
LIN {X 0.163,Y -585.316,Z 1086.521,A 0.000,B 0.000,C 90.000,E1 309.725} C_DIS
LIN {X -0.008,Y -582.147,Z 1086.515,A 0.000,B 0.000,C 90.000,E1 308.669} C_DIS
LIN {X 0.344,Y -580.360,Z 1086.512,A 0.000,B 0.000,C 90.000,E1 308.096} C_DIS
LIN {X -0.102,Y -575.531,Z 1086.504,A 0.000,B 0.000,C 90.000,E1 306.790} C_DIS
LIN {X 0.010,Y -572.319,Z 1086.500,A 0.000,B 0.000,C 90.000,E1 305.964} C_DIS
LIN {X -0.271,Y -569.476,Z 1086.496,A 0.000,B 0.000,C 90.000,E1 305.311} C_DIS
LIN {X -0.016,Y -566.733,Z 1086.493,A 0.000,B 0.000,C 90.000,E1 304.739} C_DIS
LIN {X 0.106,Y -562.678,Z 1086.489,A 0.000,B 0.000,C 90.000,E1 304.040} C_DIS
LIN {X -0.010,Y -559.224,Z 1086.486,A 0.000,B 0.000,C 90.000,E1 303.499} C_DIS
LIN {X 0.076,Y -557.085,Z 1086.485,A 0.000,B 0.000,C 90.000,E1 303.214} C_DIS
LIN {X -0.229,Y -547.936,Z 1086.478,A 0.000,B 0.000,C 90.000,E1 302.133} C_DIS
LIN {X 0.005,Y -545.377,Z 1086.476,A 0.000,B 0.000,C 90.000,E1 301.720} C_DIS
LIN {X 0.088,Y -543.466,Z 1086.474,A 0.000,B 0.000,C 90.000,E1 301.288} C_DIS
LIN {X -0.091,Y -542.965,Z 1086.473,A 0.000,B 0.000,C 90.000,E1 301.131} C_DIS
LIN {X -0.074,Y -541.683,Z 1086.471,A 0.000,B 0.000,C 90.000,E1 300.846} C_DIS
LIN {X 0.259,Y -541.184,Z 1086.471,A 0.000,B 0.000,C 90.000,E1 300.669} C_DIS
LIN {X 0.000,Y -539.895,Z 1086.467,A 0.000,B 0.000,C 90.000,E1 300.129} C_DIS
LIN {X 0.332,Y -539.358,Z 1086.465,A 0.000,B 0.000,C 90.000,E1 299.667} C_DIS
LIN {X -0.116,Y -539.401,Z 1086.464,A 0.000,B 0.000,C 90.000,E1 299.539} C_DIS
LIN {X 0.079,Y -539.078,Z 1086.461,A 0.000,B 0.000,C 90.000,E1 298.949} C_DIS
LIN {X 0.002,Y -538.925,Z 1086.456,A 0.000,B 0.000,C 90.000,E1 298.103} C_DIS
LIN {X -0.266,Y -539.527,Z 1086.440,A 0.000,B 0.000,C 90.000,E1 295.283} C_DIS
LIN {X -0.179,Y -540.111,Z 1086.431,A 0.000,B 0.000,C 90.000,E1 293.567} C_DIS
LIN {X -0.017,Y -540.620,Z 1086.421,A 0.000,B 0.000,C 90.000,E1 291.844} C_DIS
LIN {X 0.162,Y -541.039,Z 1086.412,A 0.000,B 0.000,C 90.000,E1 290.120} C_DIS
LIN {X -0.124,Y -541.171,Z 1086.406,A 0.000,B 0.000,C 90.000,E1 289.014} C_DIS
LIN {X -0.076,Y -541.055,Z 1086.399,A 0.000,B 0.000,C 90.000,E1 287.873} C_DIS
LIN {X -0.026,Y -540.904,Z 1086.393,A 0.000,B 0.000,C 90.000,E1 286.732} C_DIS
LIN {X 0.081,Y -540.567,Z 1086.385,A 0.000,B 0.000,C 90.000,E1 285.300} C_DIS
LIN {X -0.029,Y -540.136,Z 1086.379,A 0.000,B 0.000,C 90.000,E1 284.175} C_DIS
LIN {X -0.199,Y -539.534,Z 1086.371,A 0.000,B 0.000,C 90.000,E1 282.771} C_DIS
LIN {X -0.299,Y -538.691,Z 1086.361,A 0.000,B 0.000,C 90.000,E1 281.074} C_DIS
LIN {X 0.103,Y -537.814,Z 1086.352,A 0.000,B 0.000,C 90.000,E1 279.321} C_DIS
LIN {X -0.281,Y -537.082,Z 1086.344,A 0.000,B 0.000,C 90.000,E1 277.936} C_DIS
LIN {X -0.037,Y -536.128,Z 1086.333,A 0.000,B 0.000,C 90.000,E1 275.910} C_DIS
LIN {X 0.023,Y -535.201,Z 1086.323,A 0.000,B 0.000,C 90.000,E1 274.188} C_DIS
LIN {X 0.072,Y -534.490,Z 1086.315,A 0.000,B 0.000,C 90.000,E1 272.751} C_DIS
LIN {X 0.069,Y -533.583,Z 1086.304,A 0.000,B 0.000,C 90.000,E1 270.745} C_DIS
LIN {X 0.046,Y -532.819,Z 1086.296,A 0.000,B 0.000,C 90.000,E1 269.312} C_DIS
LIN {X 0.022,Y -532.020,Z 1086.288,A 0.000,B 0.000,C 90.000,E1 267.879} C_DIS
LIN {X -0.016,Y -531.198,Z 1086.280,A 0.000,B 0.000,C 90.000,E1 266.445} C_DIS
LIN {X -0.041,Y -529.841,Z 1086.269,A 0.000,B 0.000,C 90.000,E1 264.432} C_DIS
LIN {X -0.096,Y -528.594,Z 1086.261,A 0.000,B 0.000,C 90.000,E1 262.996} C_DIS
LIN {X -0.084,Y -526.387,Z 1086.250,A 0.000,B 0.000,C 90.000,E1 260.971} C_DIS
LIN {X 0.036,Y -524.623,Z 1086.240,A 0.000,B 0.000,C 90.000,E1 259.218} C_DIS
LIN {X 0.100,Y -523.411,Z 1086.234,A 0.000,B 0.000,C 90.000,E1 258.049} C_DIS
LIN {X 0.280,Y -521.426,Z 1086.222,A 0.000,B 0.000,C 90.000,E1 255.992} C_DIS
LIN {X -0.098,Y -519.971,Z 1086.214,A 0.000,B 0.000,C 90.000,E1 254.574} C_DIS
LIN {X 0.263,Y -518.140,Z 1086.205,A 0.000,B 0.000,C 90.000,E1 252.779} C_DIS
LIN {X 0.214,Y -515.911,Z 1086.193,A 0.000,B 0.000,C 90.000,E1 250.732} C_DIS
LIN {X 0.071,Y -514.679,Z 1086.187,A 0.000,B 0.000,C 90.000,E1 249.571} C_DIS
LIN {X 0.151,Y -512.459,Z 1086.177,A 0.000,B 0.000,C 90.000,E1 247.794} C_DIS
LIN {X -0.212,Y -510.489,Z 1086.169,A 0.000,B 0.000,C 90.000,E1 246.357} C_DIS
LIN {X 0.110,Y -509.156,Z 1086.164,A 0.000,B 0.000,C 90.000,E1 245.433} C_DIS
LIN {X -0.163,Y -505.852,Z 1086.152,A 0.000,B 0.000,C 90.000,E1 243.384} C_DIS
LIN {X -0.206,Y -503.348,Z 1086.144,A 0.000,B 0.000,C 90.000,E1 241.897} C_DIS
LIN {X 0.083,Y -501.295,Z 1086.137,A 0.000,B 0.000,C 90.000,E1 240.667} C_DIS
LIN {X 0.045,Y -498.159,Z 1086.127,A 0.000,B 0.000,C 90.000,E1 238.869} C_DIS
LIN {X -0.074,Y -495.443,Z 1086.119,A 0.000,B 0.000,C 90.000,E1 237.375} C_DIS
LIN {X 0.012,Y -492.033,Z 1086.109,A 0.000,B 0.000,C 90.000,E1 235.548} C_DIS
LIN {X -0.072,Y -489.043,Z 1086.100,A 0.000,B 0.000,C 90.000,E1 234.036} C_DIS
LIN {X 0.064,Y -486.653,Z 1086.093,A 0.000,B 0.000,C 90.000,E1 232.798} C_DIS
LIN {X -0.001,Y -482.832,Z 1086.083,A 0.000,B 0.000,C 90.000,E1 230.964} C_DIS
LIN {X -0.322,Y -479.517,Z 1086.075,A 0.000,B 0.000,C 90.000,E1 229.461} C_DIS
LIN {X 0.077,Y -475.727,Z 1086.064,A 0.000,B 0.000,C 90.000,E1 227.553} C_DIS
LIN {X 0.027,Y -472.190,Z 1086.054,A 0.000,B 0.000,C 90.000,E1 225.688} C_DIS
LIN {X -0.024,Y -468.158,Z 1086.042,A 0.000,B 0.000,C 90.000,E1 223.500} C_DIS
LIN {X 0.081,Y -464.542,Z 1086.031,A 0.000,B 0.000,C 90.000,E1 221.595} C_DIS
LIN {X -0.172,Y -460.913,Z 1086.021,A 0.000,B 0.000,C 90.000,E1 219.725} C_DIS
LIN {X 0.117,Y -457.929,Z 1086.012,A 0.000,B 0.000,C 90.000,E1 218.096} C_DIS
LIN {X 0.059,Y -454.969,Z 1086.003,A 0.000,B 0.000,C 90.000,E1 216.503} C_DIS
LIN {X 0.043,Y -452.081,Z 1085.994,A 0.000,B 0.000,C 90.000,E1 214.898} C_DIS
LIN {X 0.128,Y -447.912,Z 1085.981,A 0.000,B 0.000,C 90.000,E1 212.625} C_DIS
LIN {X 0.170,Y -444.413,Z 1085.971,A 0.000,B 0.000,C 90.000,E1 210.669} C_DIS
LIN {X -0.056,Y -440.549,Z 1085.958,A 0.000,B 0.000,C 90.000,E1 208.409} C_DIS
LIN {X -0.119,Y -434.668,Z 1085.936,A 0.000,B 0.000,C 90.000,E1 204.463} C_DIS
LIN {X -0.073,Y -432.869,Z 1085.928,A 0.000,B 0.000,C 90.000,E1 203.131} C_DIS
LIN {X -0.213,Y -431.832,Z 1085.923,A 0.000,B 0.000,C 90.000,E1 202.153} C_DIS
LIN {X 0.015,Y -430.845,Z 1085.916,A 0.000,B 0.000,C 90.000,E1 200.791} C_DIS
LIN {X 0.044,Y -430.721,Z 1085.912,A 0.000,B 0.000,C 90.000,E1 200.120} C_DIS
LIN {X -0.117,Y -431.072,Z 1085.906,A 0.000,B 0.000,C 90.000,E1 199.141} C_DIS
LIN {X -0.090,Y -431.731,Z 1085.903,A 0.000,B 0.000,C 90.000,E1 198.471} C_DIS
LIN {X -0.194,Y -432.770,Z 1085.899,A 0.000,B 0.000,C 90.000,E1 197.819} C_DIS
LIN {X -0.055,Y -435.350,Z 1085.893,A 0.000,B 0.000,C 90.000,E1 196.804} C_DIS
LIN {X -0.004,Y -437.542,Z 1085.890,A 0.000,B 0.000,C 90.000,E1 196.134} C_DIS
LIN {X -0.071,Y -443.473,Z 1085.881,A 0.000,B 0.000,C 90.000,E1 194.662} C_DIS
LIN {X 0.178,Y -453.785,Z 1085.869,A 0.000,B 0.000,C 90.000,E1 192.355} C_DIS
LIN {X -0.218,Y -466.659,Z 1085.855,A 0.000,B 0.000,C 90.000,E1 189.849} C_DIS
LIN {X 0.255,Y -474.919,Z 1085.846,A 0.000,B 0.000,C 90.000,E1 188.219} C_DIS
LIN {X 0.016,Y -481.383,Z 1085.839,A 0.000,B 0.000,C 90.000,E1 187.004} C_DIS
LIN {X 0.142,Y -484.558,Z 1085.836,A 0.000,B 0.000,C 90.000,E1 186.372} C_DIS
LIN {X -0.169,Y -489.945,Z 1085.830,A 0.000,B 0.000,C 90.000,E1 185.334} C_DIS
LIN {X 0.209,Y -495.992,Z 1085.823,A 0.000,B 0.000,C 90.000,E1 184.073} C_DIS
LIN {X 0.102,Y -503.453,Z 1085.814,A 0.000,B 0.000,C 90.000,E1 182.579} C_DIS
LIN {X 0.012,Y -512.283,Z 1085.805,A 0.000,B 0.000,C 90.000,E1 180.802} C_DIS
LIN {X 0.109,Y -521.092,Z 1085.795,A 0.000,B 0.000,C 90.000,E1 179.026} C_DIS
LIN {X 0.194,Y -527.677,Z 1085.787,A 0.000,B 0.000,C 90.000,E1 177.707} C_DIS
LIN {X -0.152,Y -535.594,Z 1085.779,A 0.000,B 0.000,C 90.000,E1 176.159} C_DIS
LIN {X 0.207,Y -541.979,Z 1085.771,A 0.000,B 0.000,C 90.000,E1 174.837} C_DIS
LIN {X 0.134,Y -548.372,Z 1085.764,A 0.000,B 0.000,C 90.000,E1 173.571} C_DIS
LIN {X -0.204,Y -556.048,Z 1085.756,A 0.000,B 0.000,C 90.000,E1 172.064} C_DIS
LIN {X 0.013,Y -562.144,Z 1085.749,A 0.000,B 0.000,C 90.000,E1 170.792} C_DIS
LIN {X 0.005,Y -567.470,Z 1085.743,A 0.000,B 0.000,C 90.000,E1 169.690} C_DIS
LIN {X -0.256,Y -571.963,Z 1085.737,A 0.000,B 0.000,C 90.000,E1 168.757} C_DIS
LIN {X 0.216,Y -576.364,Z 1085.732,A 0.000,B 0.000,C 90.000,E1 167.757} C_DIS
LIN {X -0.048,Y -581.189,Z 1085.726,A 0.000,B 0.000,C 90.000,E1 166.700} C_DIS
LIN {X -0.262,Y -585.848,Z 1085.720,A 0.000,B 0.000,C 90.000,E1 165.644} C_DIS
LIN {X -0.199,Y -588.154,Z 1085.717,A 0.000,B 0.000,C 90.000,E1 165.102} C_DIS
LIN {X -0.168,Y -592.485,Z 1085.711,A 0.000,B 0.000,C 90.000,E1 164.031} C_DIS
LIN {X 0.222,Y -595.516,Z 1085.707,A 0.000,B 0.000,C 90.000,E1 163.196} C_DIS
LIN {X -0.223,Y -599.361,Z 1085.701,A 0.000,B 0.000,C 90.000,E1 162.181} C_DIS
LIN {X 0.137,Y -603.031,Z 1085.695,A 0.000,B 0.000,C 90.000,E1 161.094} C_DIS
LIN {X -0.023,Y -606.440,Z 1085.689,A 0.000,B 0.000,C 90.000,E1 160.061} C_DIS
LIN {X -0.141,Y -609.673,Z 1085.683,A 0.000,B 0.000,C 90.000,E1 159.028} C_DIS
LIN {X 0.002,Y -612.762,Z 1085.678,A 0.000,B 0.000,C 90.000,E1 157.975} C_DIS
LIN {X 0.165,Y -616.410,Z 1085.671,A 0.000,B 0.000,C 90.000,E1 156.666} C_DIS
LIN {X -0.146,Y -618.574,Z 1085.666,A 0.000,B 0.000,C 90.000,E1 155.921} C_DIS
LIN {X 0.101,Y -622.551,Z 1085.658,A 0.000,B 0.000,C 90.000,E1 154.357} C_DIS
LIN {X 0.120,Y -625.738,Z 1085.651,A 0.000,B 0.000,C 90.000,E1 153.076} C_DIS
LIN {X -0.047,Y -629.441,Z 1085.642,A 0.000,B 0.000,C 90.000,E1 151.563} C_DIS
LIN {X -0.127,Y -632.814,Z 1085.634,A 0.000,B 0.000,C 90.000,E1 150.049} C_DIS
LIN {X -0.147,Y -636.081,Z 1085.625,A 0.000,B 0.000,C 90.000,E1 148.535} C_DIS
LIN {X 0.176,Y -638.696,Z 1085.618,A 0.000,B 0.000,C 90.000,E1 147.248} C_DIS
LIN {X 0.010,Y -641.219,Z 1085.611,A 0.000,B 0.000,C 90.000,E1 146.008} C_DIS
LIN {X -0.159,Y -643.198,Z 1085.606,A 0.000,B 0.000,C 90.000,E1 145.022} C_DIS
LIN {X -0.261,Y -645.586,Z 1085.599,A 0.000,B 0.000,C 90.000,E1 143.783} C_DIS
LIN {X 0.043,Y -647.917,Z 1085.592,A 0.000,B 0.000,C 90.000,E1 142.512} C_DIS
LIN {X 0.163,Y -651.723,Z 1085.581,A 0.000,B 0.000,C 90.000,E1 140.517} C_DIS
LIN {X 0.012,Y -653.735,Z 1085.575,A 0.000,B 0.000,C 90.000,E1 139.542} C_DIS
LIN {X 0.222,Y -657.673,Z 1085.564,A 0.000,B 0.000,C 90.000,E1 137.553} C_DIS
LIN {X -0.414,Y -661.300,Z 1085.555,A 0.000,B 0.000,C 90.000,E1 135.891} C_DIS
LIN {X 0.436,Y -665.325,Z 1085.545,A 0.000,B 0.000,C 90.000,E1 134.109} C_DIS
LIN {X -0.025,Y -669.586,Z 1085.536,A 0.000,B 0.000,C 90.000,E1 132.447} C_DIS
LIN {X 0.196,Y -675.104,Z 1085.524,A 0.000,B 0.000,C 90.000,E1 130.253} C_DIS
LIN {X -0.029,Y -678.708,Z 1085.516,A 0.000,B 0.000,C 90.000,E1 128.830} C_DIS
LIN {X -0.053,Y -683.105,Z 1085.506,A 0.000,B 0.000,C 90.000,E1 127.156} C_DIS
LIN {X -0.046,Y -686.165,Z 1085.500,A 0.000,B 0.000,C 90.000,E1 125.964} C_DIS
LIN {X -0.179,Y -688.465,Z 1085.495,A 0.000,B 0.000,C 90.000,E1 125.025} C_DIS
LIN {X 0.123,Y -691.884,Z 1085.487,A 0.000,B 0.000,C 90.000,E1 123.579} C_DIS
LIN {X -0.114,Y -694.791,Z 1085.480,A 0.000,B 0.000,C 90.000,E1 122.418} C_DIS
LIN {X -0.312,Y -697.585,Z 1085.474,A 0.000,B 0.000,C 90.000,E1 121.258} C_DIS
LIN {X -0.150,Y -699.108,Z 1085.470,A 0.000,B 0.000,C 90.000,E1 120.541} C_DIS
LIN {X 0.310,Y -701.175,Z 1085.463,A 0.000,B 0.000,C 90.000,E1 119.333} C_DIS
LIN {X 0.116,Y -702.545,Z 1085.457,A 0.000,B 0.000,C 90.000,E1 118.180} C_DIS
LIN {X -0.068,Y -703.810,Z 1085.449,A 0.000,B 0.000,C 90.000,E1 116.796} C_DIS
LIN {X -0.237,Y -705.017,Z 1085.441,A 0.000,B 0.000,C 90.000,E1 115.412} C_DIS
LIN {X 0.051,Y -705.167,Z 1085.440,A 0.000,B 0.000,C 90.000,E1 115.155} C_DIS
LIN {X -0.013,Y -705.195,Z 1085.437,A 0.000,B 0.000,C 90.000,E1 114.695} C_DIS
LIN {X 0.268,Y -704.758,Z 1085.435,A 0.000,B 0.000,C 90.000,E1 114.207} C_DIS
LIN {X -0.089,Y -704.462,Z 1085.433,A 0.000,B 0.000,C 90.000,E1 114.003} C_DIS
LIN {X 0.193,Y -702.881,Z 1085.431,A 0.000,B 0.000,C 90.000,E1 113.515} C_DIS
LIN {X -0.451,Y -701.888,Z 1085.429,A 0.000,B 0.000,C 90.000,E1 113.334} C_DIS
LIN {X 0.115,Y -698.269,Z 1085.427,A 0.000,B 0.000,C 90.000,E1 112.823} C_DIS
LIN {X -0.025,Y -697.236,Z 1085.426,A 0.000,B 0.000,C 90.000,E1 112.717} C_DIS
LIN {X 0.106,Y -695.701,Z 1085.426,A 0.000,B 0.000,C 90.000,E1 112.589} C_DIS
LIN {X 0.061,Y -691.180,Z 1085.424,A 0.000,B 0.000,C 90.000,E1 112.386} C_DIS
LIN {X 0.314,Y -686.128,Z 1085.423,A 0.000,B 0.000,C 90.000,E1 112.153} C_DIS
LIN {X 0.095,Y -682.468,Z 1085.423,A 0.000,B 0.000,C 90.000,E1 112.099} C_DIS
LIN {X -0.033,Y -675.804,Z 1085.422,A 0.000,B 0.000,C 90.000,E1 112.025} C_DIS
LIN {X -0.077,Y -605.182,Z 1085.422,A 0.000,B 0.000,C 90.000,E1 112.025} C_DIS
LIN {X 0.177,Y -601.872,Z 1085.422,A 0.000,B 0.000,C 90.000,E1 111.844} C_DIS
LIN {X -0.287,Y -596.359,Z 1085.420,A 0.000,B 0.000,C 90.000,E1 111.535} C_DIS
LIN {X -0.211,Y -584.469,Z 1085.414,A 0.000,B 0.000,C 90.000,E1 110.556} C_DIS
LIN {X 0.158,Y -576.077,Z 1085.410,A 0.000,B 0.000,C 90.000,E1 109.812} C_DIS
LIN {X -0.267,Y -570.057,Z 1085.408,A 0.000,B 0.000,C 90.000,E1 109.396} C_DIS
LIN {X -0.095,Y -568.580,Z 1085.407,A 0.000,B 0.000,C 90.000,E1 109.268} C_DIS
LIN {X 0.216,Y -560.232,Z 1085.404,A 0.000,B 0.000,C 90.000,E1 108.725} C_DIS
LIN {X 0.186,Y -553.951,Z 1085.402,A 0.000,B 0.000,C 90.000,E1 108.362} C_DIS
LIN {X 0.252,Y -549.545,Z 1085.401,A 0.000,B 0.000,C 90.000,E1 108.055} C_DIS
LIN {X 0.003,Y -547.904,Z 1085.399,A 0.000,B 0.000,C 90.000,E1 107.873} C_DIS
LIN {X -0.028,Y -547.892,Z 1085.399,A 0.000,B 0.000,C 90.000,E1 107.873} C_DIS
LIN {X -0.155,Y -547.655,Z 1085.398,A 0.000,B 0.000,C 90.000,E1 107.692} C_DIS
LIN {X -0.075,Y -547.631,Z 1085.396,A 0.000,B 0.000,C 90.000,E1 107.275} C_DIS
LIN {X -0.267,Y -548.706,Z 1085.387,A 0.000,B 0.000,C 90.000,E1 105.607} C_DIS
LIN {X 0.198,Y -550.089,Z 1085.376,A 0.000,B 0.000,C 90.000,E1 103.592} C_DIS
LIN {X 0.147,Y -552.325,Z 1085.362,A 0.000,B 0.000,C 90.000,E1 101.074} C_DIS
LIN {X -0.062,Y -554.634,Z 1085.349,A 0.000,B 0.000,C 90.000,E1 98.859} C_DIS
LIN {X -0.068,Y -556.156,Z 1085.341,A 0.000,B 0.000,C 90.000,E1 97.466} C_DIS
LIN {X -0.187,Y -557.724,Z 1085.334,A 0.000,B 0.000,C 90.000,E1 96.087} C_DIS
LIN {X 0.212,Y -558.763,Z 1085.328,A 0.000,B 0.000,C 90.000,E1 94.935} C_DIS
LIN {X 0.065,Y -559.669,Z 1085.321,A 0.000,B 0.000,C 90.000,E1 93.841} C_DIS
LIN {X 0.163,Y -560.855,Z 1085.311,A 0.000,B 0.000,C 90.000,E1 91.892} C_DIS
LIN {X 0.195,Y -561.645,Z 1085.301,A 0.000,B 0.000,C 90.000,E1 90.229} C_DIS
LIN {X 0.230,Y -562.324,Z 1085.292,A 0.000,B 0.000,C 90.000,E1 88.568} C_DIS
LIN {X -0.146,Y -563.106,Z 1085.281,A 0.000,B 0.000,C 90.000,E1 86.674} C_DIS
LIN {X -0.178,Y -563.630,Z 1085.274,A 0.000,B 0.000,C 90.000,E1 85.298} C_DIS
LIN {X -0.258,Y -564.025,Z 1085.268,A 0.000,B 0.000,C 90.000,E1 84.204} C_DIS
LIN {X -0.090,Y -564.522,Z 1085.259,A 0.000,B 0.000,C 90.000,E1 82.534} C_DIS
LIN {X 0.078,Y -565.022,Z 1085.251,A 0.000,B 0.000,C 90.000,E1 81.141} C_DIS
LIN {X 0.045,Y -565.784,Z 1085.240,A 0.000,B 0.000,C 90.000,E1 79.218} C_DIS
LIN {X -0.320,Y -566.387,Z 1085.233,A 0.000,B 0.000,C 90.000,E1 77.881} C_DIS
LIN {X -0.089,Y -567.371,Z 1085.222,A 0.000,B 0.000,C 90.000,E1 75.936} C_DIS
LIN {X -0.011,Y -568.437,Z 1085.213,A 0.000,B 0.000,C 90.000,E1 74.283} C_DIS
LIN {X 0.029,Y -569.898,Z 1085.202,A 0.000,B 0.000,C 90.000,E1 72.362} C_DIS
LIN {X -0.061,Y -571.232,Z 1085.193,A 0.000,B 0.000,C 90.000,E1 70.732} C_DIS
LIN {X 0.088,Y -572.189,Z 1085.187,A 0.000,B 0.000,C 90.000,E1 69.625} C_DIS
LIN {X 0.046,Y -573.083,Z 1085.181,A 0.000,B 0.000,C 90.000,E1 68.539} C_DIS
LIN {X -0.112,Y -574.495,Z 1085.172,A 0.000,B 0.000,C 90.000,E1 66.922} C_DIS
LIN {X -0.005,Y -575.713,Z 1085.163,A 0.000,B 0.000,C 90.000,E1 65.281} C_DIS
LIN {X 0.130,Y -576.816,Z 1085.154,A 0.000,B 0.000,C 90.000,E1 63.640} C_DIS
LIN {X -0.125,Y -578.014,Z 1085.143,A 0.000,B 0.000,C 90.000,E1 61.769} C_DIS
LIN {X 0.067,Y -578.949,Z 1085.134,A 0.000,B 0.000,C 90.000,E1 60.127} C_DIS
LIN {X -0.227,Y -579.808,Z 1085.125,A 0.000,B 0.000,C 90.000,E1 58.535} C_DIS
LIN {X -0.041,Y -580.743,Z 1085.115,A 0.000,B 0.000,C 90.000,E1 56.628} C_DIS
LIN {X 0.146,Y -581.322,Z 1085.107,A 0.000,B 0.000,C 90.000,E1 55.261} C_DIS
LIN {X 0.027,Y -581.931,Z 1085.098,A 0.000,B 0.000,C 90.000,E1 53.657} C_DIS
LIN {X 0.259,Y -582.203,Z 1085.092,A 0.000,B 0.000,C 90.000,E1 52.557} C_DIS
LIN {X -0.032,Y -582.325,Z 1085.088,A 0.000,B 0.000,C 90.000,E1 51.778} C_DIS
LIN {X -0.068,Y -582.191,Z 1085.080,A 0.000,B 0.000,C 90.000,E1 50.436} C_DIS
LIN {X -0.272,Y -581.965,Z 1085.074,A 0.000,B 0.000,C 90.000,E1 49.380} C_DIS
LIN {X 0.340,Y -581.579,Z 1085.068,A 0.000,B 0.000,C 90.000,E1 48.243} C_DIS
LIN {X -0.022,Y -580.905,Z 1085.059,A 0.000,B 0.000,C 90.000,E1 46.662} C_DIS
LIN {X 0.144,Y -580.239,Z 1085.053,A 0.000,B 0.000,C 90.000,E1 45.567} C_DIS
LIN {X 0.154,Y -579.613,Z 1085.049,A 0.000,B 0.000,C 90.000,E1 44.757} C_DIS
LIN {X 0.156,Y -578.826,Z 1085.044,A 0.000,B 0.000,C 90.000,E1 43.947} C_DIS
LIN {X 0.291,Y -577.600,Z 1085.038,A 0.000,B 0.000,C 90.000,E1 42.852} C_DIS
LIN {X 0.119,Y -575.714,Z 1085.031,A 0.000,B 0.000,C 90.000,E1 41.515} C_DIS
LIN {X 0.264,Y -575.325,Z 1085.029,A 0.000,B 0.000,C 90.000,E1 41.229} C_DIS
LIN {X -0.035,Y -573.458,Z 1085.023,A 0.000,B 0.000,C 90.000,E1 40.172} C_DIS
LIN {X 0.083,Y -571.319,Z 1085.017,A 0.000,B 0.000,C 90.000,E1 39.072} C_DIS
LIN {X 0.172,Y -568.868,Z 1085.011,A 0.000,B 0.000,C 90.000,E1 37.971} C_DIS
LIN {X -0.149,Y -568.217,Z 1085.010,A 0.000,B 0.000,C 90.000,E1 37.729} C_DIS
LIN {X 0.338,Y -565.045,Z 1085.004,A 0.000,B 0.000,C 90.000,E1 36.583} C_DIS
LIN {X -0.117,Y -562.386,Z 1084.999,A 0.000,B 0.000,C 90.000,E1 35.804} C_DIS
LIN {X -0.044,Y -558.067,Z 1084.993,A 0.000,B 0.000,C 90.000,E1 34.692} C_DIS
LIN {X -0.105,Y -554.565,Z 1084.988,A 0.000,B 0.000,C 90.000,E1 33.865} C_DIS
LIN {X -0.087,Y -551.297,Z 1084.984,A 0.000,B 0.000,C 90.000,E1 33.166} C_DIS
LIN {X -0.104,Y -547.769,Z 1084.980,A 0.000,B 0.000,C 90.000,E1 32.467} C_DIS
LIN {X 0.042,Y -542.622,Z 1084.975,A 0.000,B 0.000,C 90.000,E1 31.465} C_DIS
LIN {X 0.122,Y -538.633,Z 1084.971,A 0.000,B 0.000,C 90.000,E1 30.747} C_DIS
LIN {X -0.166,Y -533.549,Z 1084.966,A 0.000,B 0.000,C 90.000,E1 29.922} C_DIS
LIN {X -0.166,Y -528.813,Z 1084.962,A 0.000,B 0.000,C 90.000,E1 29.205} C_DIS
LIN {X -0.052,Y -524.754,Z 1084.959,A 0.000,B 0.000,C 90.000,E1 28.615} C_DIS
LIN {X 0.030,Y -520.408,Z 1084.956,A 0.000,B 0.000,C 90.000,E1 28.025} C_DIS
LIN {X 0.197,Y -513.356,Z 1084.951,A 0.000,B 0.000,C 90.000,E1 27.129} C_DIS
LIN {X 0.052,Y -506.881,Z 1084.947,A 0.000,B 0.000,C 90.000,E1 26.411} C_DIS
LIN {X 0.045,Y -501.654,Z 1084.944,A 0.000,B 0.000,C 90.000,E1 25.848} C_DIS
LIN {X -0.265,Y -492.203,Z 1084.938,A 0.000,B 0.000,C 90.000,E1 24.899} C_DIS
LIN {X -0.202,Y -483.775,Z 1084.934,A 0.000,B 0.000,C 90.000,E1 24.079} C_DIS
LIN {X -0.151,Y -475.052,Z 1084.929,A 0.000,B 0.000,C 90.000,E1 23.259} C_DIS
LIN {X 0.098,Y -470.649,Z 1084.927,A 0.000,B 0.000,C 90.000,E1 22.823} C_DIS
LIN {X 0.128,Y -457.268,Z 1084.921,A 0.000,B 0.000,C 90.000,E1 21.663} C_DIS
LIN {X -0.252,Y -448.189,Z 1084.916,A 0.000,B 0.000,C 90.000,E1 20.918} C_DIS
LIN {X -0.088,Y -431.956,Z 1084.908,A 0.000,B 0.000,C 90.000,E1 19.396} C_DIS
LIN {X -0.096,Y -416.268,Z 1084.899,A 0.000,B 0.000,C 90.000,E1 17.764} C_DIS
LIN {X 0.191,Y -405.445,Z 1084.891,A 0.000,B 0.000,C 90.000,E1 16.441} C_DIS
LIN {X 0.046,Y -399.067,Z 1084.887,A 0.000,B 0.000,C 90.000,E1 15.607} C_DIS
LIN {X 0.127,Y -396.776,Z 1084.885,A 0.000,B 0.000,C 90.000,E1 15.245} C_DIS
LIN {X 0.137,Y -394.549,Z 1084.883,A 0.000,B 0.000,C 90.000,E1 14.828} C_DIS
LIN {X 0.028,Y -392.754,Z 1084.880,A 0.000,B 0.000,C 90.000,E1 14.300} C_DIS
LIN {X 0.004,Y -392.083,Z 1084.877,A 0.000,B 0.000,C 90.000,E1 13.772} C_DIS
LIN {X -0.003,Y -392.165,Z 1084.873,A 0.000,B 0.000,C 90.000,E1 13.063} C_DIS
LIN {X -0.061,Y -393.269,Z 1084.867,A 0.000,B 0.000,C 90.000,E1 12.007} C_DIS
LIN {X 0.103,Y -398.693,Z 1084.849,A 0.000,B 0.000,C 90.000,E1 8.803} C_DIS
LIN {X -0.094,Y -404.830,Z 1084.833,A 0.000,B 0.000,C 90.000,E1 6.030} C_DIS
LIN {X -0.129,Y -407.119,Z 1084.828,A 0.000,B 0.000,C 90.000,E1 4.992} C_DIS
LIN {X -0.152,Y -409.359,Z 1084.824,A 0.000,B 0.000,C 90.000,E1 4.302} C_DIS
LIN {X 0.172,Y -412.841,Z 1084.820,A 0.000,B 0.000,C 90.000,E1 3.612} C_DIS
LIN {X 0.062,Y -416.624,Z 1084.818,A 0.000,B 0.000,C 90.000,E1 3.212} C_DIS
LIN {X 0.113,Y -422.165,Z 1084.815,A 0.000,B 0.000,C 90.000,E1 2.751} C_DIS
LIN {X 0.161,Y -427.532,Z 1084.814,A 0.000,B 0.000,C 90.000,E1 2.407} C_DIS
LIN {X -0.052,Y -447.140,Z 1084.806,A 0.000,B 0.000,C 90.000,E1 1.146} C_DIS
LIN {X -0.138,Y -461.796,Z 1084.801,A 0.000,B 0.000,C 90.000,E1 0.229} C_DIS
LIN {X 0.028,Y -473.412,Z 1084.797,A 0.000,B 0.000,C 90.000,E1 359.484} C_DIS
LIN {X -0.182,Y -484.808,Z 1084.793,A 0.000,B 0.000,C 90.000,E1 358.797} C_DIS
LIN {X 0.149,Y -491.197,Z 1084.791,A 0.000,B 0.000,C 90.000,E1 358.339} C_DIS
LIN {X 0.025,Y -502.267,Z 1084.787,A 0.000,B 0.000,C 90.000,E1 357.593} C_DIS
LIN {X 0.127,Y -511.339,Z 1084.783,A 0.000,B 0.000,C 90.000,E1 356.906} C_DIS
LIN {X 0.102,Y -515.853,Z 1084.781,A 0.000,B 0.000,C 90.000,E1 356.560} C_DIS
LIN {X -0.058,Y -522.873,Z 1084.778,A 0.000,B 0.000,C 90.000,E1 355.988} C_DIS
LIN {X 0.000,Y -528.277,Z 1084.775,A 0.000,B 0.000,C 90.000,E1 355.469} C_DIS
LIN {X 0.014,Y -532.374,Z 1084.773,A 0.000,B 0.000,C 90.000,E1 355.065} C_DIS
LIN {X 0.072,Y -539.625,Z 1084.768,A 0.000,B 0.000,C 90.000,E1 354.261} C_DIS
LIN {X -0.127,Y -545.395,Z 1084.764,A 0.000,B 0.000,C 90.000,E1 353.571} C_DIS
LIN {X 0.234,Y -548.733,Z 1084.762,A 0.000,B 0.000,C 90.000,E1 353.109} C_DIS
LIN {X 0.181,Y -553.485,Z 1084.758,A 0.000,B 0.000,C 90.000,E1 352.413} C_DIS
LIN {X 0.092,Y -557.813,Z 1084.754,A 0.000,B 0.000,C 90.000,E1 351.724} C_DIS
LIN {X 0.121,Y -561.616,Z 1084.750,A 0.000,B 0.000,C 90.000,E1 351.027} C_DIS
LIN {X 0.182,Y -565.133,Z 1084.746,A 0.000,B 0.000,C 90.000,E1 350.330} C_DIS
LIN {X 0.136,Y -568.935,Z 1084.742,A 0.000,B 0.000,C 90.000,E1 349.511} C_DIS
LIN {X 0.020,Y -572.379,Z 1084.737,A 0.000,B 0.000,C 90.000,E1 348.701} C_DIS
LIN {X 0.045,Y -575.630,Z 1084.733,A 0.000,B 0.000,C 90.000,E1 347.881} C_DIS
LIN {X -0.246,Y -579.693,Z 1084.727,A 0.000,B 0.000,C 90.000,E1 346.825} C_DIS
LIN {X 0.121,Y -585.323,Z 1084.718,A 0.000,B 0.000,C 90.000,E1 345.172} C_DIS
LIN {X -0.215,Y -589.663,Z 1084.710,A 0.000,B 0.000,C 90.000,E1 343.866} C_DIS
LIN {X -0.002,Y -592.994,Z 1084.704,A 0.000,B 0.000,C 90.000,E1 342.779} C_DIS
LIN {X -0.035,Y -597.021,Z 1084.697,A 0.000,B 0.000,C 90.000,E1 341.456} C_DIS
LIN {X 0.288,Y -599.856,Z 1084.691,A 0.000,B 0.000,C 90.000,E1 340.369} C_DIS
LIN {X 0.082,Y -602.511,Z 1084.685,A 0.000,B 0.000,C 90.000,E1 339.337} C_DIS
LIN {X 0.125,Y -604.868,Z 1084.679,A 0.000,B 0.000,C 90.000,E1 338.284} C_DIS
LIN {X 0.263,Y -606.452,Z 1084.675,A 0.000,B 0.000,C 90.000,E1 337.486} C_DIS
LIN {X -0.198,Y -608.327,Z 1084.669,A 0.000,B 0.000,C 90.000,E1 336.485} C_DIS
LIN {X 0.173,Y -609.916,Z 1084.664,A 0.000,B 0.000,C 90.000,E1 335.409} C_DIS
LIN {X -0.206,Y -611.015,Z 1084.659,A 0.000,B 0.000,C 90.000,E1 334.665} C_DIS
LIN {X 0.164,Y -612.563,Z 1084.652,A 0.000,B 0.000,C 90.000,E1 333.332} C_DIS
LIN {X 0.069,Y -613.309,Z 1084.648,A 0.000,B 0.000,C 90.000,E1 332.564} C_DIS
LIN {X 0.238,Y -614.134,Z 1084.642,A 0.000,B 0.000,C 90.000,E1 331.513} C_DIS
LIN {X -0.110,Y -614.627,Z 1084.636,A 0.000,B 0.000,C 90.000,E1 330.511} C_DIS
LIN {X -0.195,Y -614.853,Z 1084.632,A 0.000,B 0.000,C 90.000,E1 329.744} C_DIS
LIN {X 0.026,Y -614.771,Z 1084.628,A 0.000,B 0.000,C 90.000,E1 328.948} C_DIS
LIN {X 0.010,Y -614.276,Z 1084.622,A 0.000,B 0.000,C 90.000,E1 327.916} C_DIS
LIN {X 0.263,Y -613.902,Z 1084.619,A 0.000,B 0.000,C 90.000,E1 327.375} C_DIS
LIN {X -0.096,Y -612.897,Z 1084.613,A 0.000,B 0.000,C 90.000,E1 326.373} C_DIS
LIN {X -0.063,Y -610.863,Z 1084.604,A 0.000,B 0.000,C 90.000,E1 324.815} C_DIS
LIN {X -0.147,Y -608.375,Z 1084.594,A 0.000,B 0.000,C 90.000,E1 323.004} C_DIS
LIN {X -0.049,Y -606.014,Z 1084.584,A 0.000,B 0.000,C 90.000,E1 321.170} C_DIS
LIN {X -0.263,Y -604.250,Z 1084.576,A 0.000,B 0.000,C 90.000,E1 319.622} C_DIS
LIN {X 0.271,Y -602.460,Z 1084.567,A 0.000,B 0.000,C 90.000,E1 318.000} C_DIS
LIN {X 0.102,Y -601.402,Z 1084.563,A 0.000,B 0.000,C 90.000,E1 317.229} C_DIS
LIN {X -0.105,Y -600.903,Z 1084.561,A 0.000,B 0.000,C 90.000,E1 316.986} C_DIS
LIN {X 0.127,Y -600.635,Z 1084.560,A 0.000,B 0.000,C 90.000,E1 316.701} C_DIS
LIN {X -0.291,Y -599.675,Z 1084.557,A 0.000,B 0.000,C 90.000,E1 316.215} C_DIS
LIN {X 0.136,Y -598.942,Z 1084.554,A 0.000,B 0.000,C 90.000,E1 315.648} C_DIS
LIN {X -0.081,Y -597.615,Z 1084.549,A 0.000,B 0.000,C 90.000,E1 314.879} C_DIS
LIN {X -0.132,Y -595.327,Z 1084.541,A 0.000,B 0.000,C 90.000,E1 313.299} C_DIS
LIN {X -0.029,Y -592.338,Z 1084.530,A 0.000,B 0.000,C 90.000,E1 311.434} C_DIS
LIN {X 0.103,Y -590.087,Z 1084.523,A 0.000,B 0.000,C 90.000,E1 310.092} C_DIS
LIN {X 0.056,Y -589.135,Z 1084.520,A 0.000,B 0.000,C 90.000,E1 309.564} C_DIS
LIN {X 0.000,Y -587.950,Z 1084.517,A 0.000,B 0.000,C 90.000,E1 309.036} C_DIS
LIN {X -0.315,Y -584.476,Z 1084.510,A 0.000,B 0.000,C 90.000,E1 307.729} C_DIS
LIN {X -0.050,Y -581.172,Z 1084.504,A 0.000,B 0.000,C 90.000,E1 306.629} C_DIS
LIN {X 0.284,Y -577.409,Z 1084.498,A 0.000,B 0.000,C 90.000,E1 305.518} C_DIS
LIN {X -0.203,Y -575.452,Z 1084.495,A 0.000,B 0.000,C 90.000,E1 305.025} C_DIS
LIN {X 0.006,Y -572.605,Z 1084.491,A 0.000,B 0.000,C 90.000,E1 304.326} C_DIS
LIN {X 0.052,Y -570.592,Z 1084.489,A 0.000,B 0.000,C 90.000,E1 303.913} C_DIS
LIN {X 0.087,Y -568.510,Z 1084.486,A 0.000,B 0.000,C 90.000,E1 303.499} C_DIS
LIN {X -0.085,Y -564.583,Z 1084.482,A 0.000,B 0.000,C 90.000,E1 302.832} C_DIS
LIN {X -0.081,Y -561.542,Z 1084.480,A 0.000,B 0.000,C 90.000,E1 302.418} C_DIS
LIN {X -0.199,Y -556.878,Z 1084.477,A 0.000,B 0.000,C 90.000,E1 301.878} C_DIS
LIN {X -0.090,Y -550.569,Z 1084.473,A 0.000,B 0.000,C 90.000,E1 301.180} C_DIS
LIN {X 0.026,Y -547.202,Z 1084.471,A 0.000,B 0.000,C 90.000,E1 300.747} C_DIS
LIN {X 0.144,Y -544.642,Z 1084.469,A 0.000,B 0.000,C 90.000,E1 300.335} C_DIS
LIN {X -0.052,Y -543.252,Z 1084.467,A 0.000,B 0.000,C 90.000,E1 300.079} C_DIS
LIN {X -0.293,Y -541.093,Z 1084.464,A 0.000,B 0.000,C 90.000,E1 299.539} C_DIS
LIN {X 0.043,Y -540.701,Z 1084.462,A 0.000,B 0.000,C 90.000,E1 299.077} C_DIS
LIN {X -0.221,Y -540.227,Z 1084.460,A 0.000,B 0.000,C 90.000,E1 298.821} C_DIS
LIN {X -0.097,Y -540.296,Z 1084.458,A 0.000,B 0.000,C 90.000,E1 298.359} C_DIS
LIN {X 0.114,Y -539.681,Z 1084.456,A 0.000,B 0.000,C 90.000,E1 298.052} C_DIS
LIN {X -0.165,Y -539.439,Z 1084.453,A 0.000,B 0.000,C 90.000,E1 297.513} C_DIS
LIN {X 0.110,Y -539.827,Z 1084.440,A 0.000,B 0.000,C 90.000,E1 295.207} C_DIS
LIN {X -0.022,Y -540.320,Z 1084.431,A 0.000,B 0.000,C 90.000,E1 293.515} C_DIS
LIN {X 0.152,Y -540.799,Z 1084.421,A 0.000,B 0.000,C 90.000,E1 291.791} C_DIS
LIN {X -0.167,Y -541.271,Z 1084.412,A 0.000,B 0.000,C 90.000,E1 290.120} C_DIS
LIN {X 0.061,Y -541.408,Z 1084.405,A 0.000,B 0.000,C 90.000,E1 288.960} C_DIS
LIN {X -0.111,Y -541.365,Z 1084.401,A 0.000,B 0.000,C 90.000,E1 288.127} C_DIS
LIN {X 0.173,Y -541.177,Z 1084.393,A 0.000,B 0.000,C 90.000,E1 286.677} C_DIS
LIN {X 0.290,Y -540.857,Z 1084.385,A 0.000,B 0.000,C 90.000,E1 285.245} C_DIS
LIN {X -0.194,Y -540.219,Z 1084.375,A 0.000,B 0.000,C 90.000,E1 283.592} C_DIS
LIN {X 0.285,Y -539.572,Z 1084.368,A 0.000,B 0.000,C 90.000,E1 282.119} C_DIS
LIN {X 0.106,Y -538.833,Z 1084.360,A 0.000,B 0.000,C 90.000,E1 280.715} C_DIS
LIN {X -0.122,Y -537.953,Z 1084.350,A 0.000,B 0.000,C 90.000,E1 279.029} C_DIS
LIN {X 0.041,Y -537.388,Z 1084.344,A 0.000,B 0.000,C 90.000,E1 277.871} C_DIS
LIN {X 0.172,Y -536.542,Z 1084.334,A 0.000,B 0.000,C 90.000,E1 276.144} C_DIS
LIN {X -0.242,Y -535.648,Z 1084.325,A 0.000,B 0.000,C 90.000,E1 274.473} C_DIS
LIN {X -0.189,Y -534.901,Z 1084.317,A 0.000,B 0.000,C 90.000,E1 273.037} C_DIS
LIN {X -0.185,Y -533.975,Z 1084.306,A 0.000,B 0.000,C 90.000,E1 271.031} C_DIS
LIN {X -0.196,Y -533.357,Z 1084.299,A 0.000,B 0.000,C 90.000,E1 269.885} C_DIS
LIN {X -0.218,Y -532.742,Z 1084.293,A 0.000,B 0.000,C 90.000,E1 268.740} C_DIS
LIN {X -0.259,Y -531.753,Z 1084.283,A 0.000,B 0.000,C 90.000,E1 267.020} C_DIS
LIN {X 0.275,Y -531.068,Z 1084.277,A 0.000,B 0.000,C 90.000,E1 265.812} C_DIS
LIN {X 0.252,Y -530.047,Z 1084.269,A 0.000,B 0.000,C 90.000,E1 264.375} C_DIS
LIN {X 0.263,Y -528.796,Z 1084.261,A 0.000,B 0.000,C 90.000,E1 262.932} C_DIS
LIN {X 0.211,Y -526.629,Z 1084.250,A 0.000,B 0.000,C 90.000,E1 260.914} C_DIS
LIN {X -0.202,Y -525.143,Z 1084.242,A 0.000,B 0.000,C 90.000,E1 259.511} C_DIS
LIN {X -0.114,Y -523.628,Z 1084.234,A 0.000,B 0.000,C 90.000,E1 258.049} C_DIS
LIN {X -0.057,Y -521.933,Z 1084.224,A 0.000,B 0.000,C 90.000,E1 256.297} C_DIS
LIN {X 0.199,Y -520.144,Z 1084.214,A 0.000,B 0.000,C 90.000,E1 254.519} C_DIS
LIN {X 0.064,Y -518.332,Z 1084.204,A 0.000,B 0.000,C 90.000,E1 252.779} C_DIS
LIN {X -0.111,Y -516.444,Z 1084.195,A 0.000,B 0.000,C 90.000,E1 251.040} C_DIS
LIN {X -0.119,Y -514.850,Z 1084.187,A 0.000,B 0.000,C 90.000,E1 249.571} C_DIS
LIN {X -0.035,Y -512.621,Z 1084.177,A 0.000,B 0.000,C 90.000,E1 247.794} C_DIS
LIN {X 0.073,Y -510.610,Z 1084.168,A 0.000,B 0.000,C 90.000,E1 246.305} C_DIS
LIN {X 0.141,Y -509.284,Z 1084.164,A 0.000,B 0.000,C 90.000,E1 245.409} C_DIS
LIN {X 0.027,Y -506.458,Z 1084.154,A 0.000,B 0.000,C 90.000,E1 243.640} C_DIS
LIN {X 0.057,Y -505.011,Z 1084.149,A 0.000,B 0.000,C 90.000,E1 242.743} C_DIS
LIN {X -0.006,Y -502.494,Z 1084.140,A 0.000,B 0.000,C 90.000,E1 241.257} C_DIS
LIN {X -0.017,Y -499.371,Z 1084.130,A 0.000,B 0.000,C 90.000,E1 239.459} C_DIS
LIN {X 0.047,Y -496.683,Z 1084.122,A 0.000,B 0.000,C 90.000,E1 237.946} C_DIS
LIN {X 0.165,Y -493.868,Z 1084.114,A 0.000,B 0.000,C 90.000,E1 236.421} C_DIS
LIN {X -0.016,Y -491.550,Z 1084.107,A 0.000,B 0.000,C 90.000,E1 235.229} C_DIS
LIN {X 0.170,Y -489.145,Z 1084.100,A 0.000,B 0.000,C 90.000,E1 233.989} C_DIS
LIN {X 0.207,Y -486.748,Z 1084.093,A 0.000,B 0.000,C 90.000,E1 232.763} C_DIS
LIN {X -0.149,Y -482.888,Z 1084.083,A 0.000,B 0.000,C 90.000,E1 230.964} C_DIS
LIN {X 0.012,Y -478.932,Z 1084.073,A 0.000,B 0.000,C 90.000,E1 229.094} C_DIS
LIN {X 0.144,Y -474.561,Z 1084.061,A 0.000,B 0.000,C 90.000,E1 226.905} C_DIS
LIN {X -0.175,Y -470.454,Z 1084.049,A 0.000,B 0.000,C 90.000,E1 224.757} C_DIS
LIN {X -0.086,Y -467.592,Z 1084.040,A 0.000,B 0.000,C 90.000,E1 223.176} C_DIS
LIN {X -0.057,Y -464.570,Z 1084.031,A 0.000,B 0.000,C 90.000,E1 221.595} C_DIS
LIN {X 0.085,Y -460.320,Z 1084.019,A 0.000,B 0.000,C 90.000,E1 219.358} C_DIS
LIN {X -0.019,Y -457.905,Z 1084.012,A 0.000,B 0.000,C 90.000,E1 218.096} C_DIS
LIN {X 0.016,Y -454.303,Z 1084.001,A 0.000,B 0.000,C 90.000,E1 216.171} C_DIS
LIN {X -0.094,Y -451.920,Z 1083.994,A 0.000,B 0.000,C 90.000,E1 214.898} C_DIS
LIN {X -0.013,Y -447.703,Z 1083.981,A 0.000,B 0.000,C 90.000,E1 212.625} C_DIS
LIN {X 0.026,Y -444.176,Z 1083.970,A 0.000,B 0.000,C 90.000,E1 210.669} C_DIS
LIN {X 0.181,Y -440.198,Z 1083.958,A 0.000,B 0.000,C 90.000,E1 208.359} C_DIS
LIN {X -0.190,Y -436.389,Z 1083.945,A 0.000,B 0.000,C 90.000,E1 206.104} C_DIS
LIN {X -0.105,Y -434.159,Z 1083.936,A 0.000,B 0.000,C 90.000,E1 204.439} C_DIS
LIN {X -0.210,Y -431.515,Z 1083.925,A 0.000,B 0.000,C 90.000,E1 202.461} C_DIS
LIN {X -0.176,Y -430.054,Z 1083.915,A 0.000,B 0.000,C 90.000,E1 200.791} C_DIS
LIN {X 0.060,Y -429.802,Z 1083.910,A 0.000,B 0.000,C 90.000,E1 199.758} C_DIS
LIN {X 0.081,Y -429.952,Z 1083.906,A 0.000,B 0.000,C 90.000,E1 199.087} C_DIS
LIN {X 0.102,Y -430.495,Z 1083.902,A 0.000,B 0.000,C 90.000,E1 198.417} C_DIS
LIN {X -0.009,Y -431.448,Z 1083.899,A 0.000,B 0.000,C 90.000,E1 197.764} C_DIS
LIN {X -0.201,Y -432.072,Z 1083.897,A 0.000,B 0.000,C 90.000,E1 197.457} C_DIS
LIN {X 0.241,Y -433.705,Z 1083.893,A 0.000,B 0.000,C 90.000,E1 196.732} C_DIS
LIN {X -0.145,Y -436.384,Z 1083.889,A 0.000,B 0.000,C 90.000,E1 195.953} C_DIS
LIN {X 0.176,Y -441.694,Z 1083.881,A 0.000,B 0.000,C 90.000,E1 194.592} C_DIS
LIN {X -0.134,Y -452.071,Z 1083.869,A 0.000,B 0.000,C 90.000,E1 192.355} C_DIS
LIN {X 0.173,Y -459.215,Z 1083.861,A 0.000,B 0.000,C 90.000,E1 190.894} C_DIS
LIN {X 0.203,Y -467.514,Z 1083.852,A 0.000,B 0.000,C 90.000,E1 189.321} C_DIS
LIN {X 0.115,Y -474.927,Z 1083.844,A 0.000,B 0.000,C 90.000,E1 187.936} C_DIS
LIN {X 0.225,Y -480.680,Z 1083.838,A 0.000,B 0.000,C 90.000,E1 186.834} C_DIS
LIN {X 0.205,Y -485.418,Z 1083.833,A 0.000,B 0.000,C 90.000,E1 185.910} C_DIS
LIN {X -0.138,Y -490.875,Z 1083.827,A 0.000,B 0.000,C 90.000,E1 184.878} C_DIS
LIN {X 0.122,Y -496.220,Z 1083.821,A 0.000,B 0.000,C 90.000,E1 183.784} C_DIS
LIN {X -0.204,Y -503.042,Z 1083.814,A 0.000,B 0.000,C 90.000,E1 182.465} C_DIS
LIN {X -0.007,Y -511.215,Z 1083.804,A 0.000,B 0.000,C 90.000,E1 180.802} C_DIS
LIN {X -0.223,Y -520.859,Z 1083.794,A 0.000,B 0.000,C 90.000,E1 178.912} C_DIS
LIN {X 0.102,Y -528.199,Z 1083.786,A 0.000,B 0.000,C 90.000,E1 177.421} C_DIS
LIN {X -0.231,Y -534.732,Z 1083.779,A 0.000,B 0.000,C 90.000,E1 176.159} C_DIS
LIN {X 0.113,Y -541.209,Z 1083.771,A 0.000,B 0.000,C 90.000,E1 174.837} C_DIS
LIN {X 0.026,Y -547.640,Z 1083.764,A 0.000,B 0.000,C 90.000,E1 173.571} C_DIS
LIN {X -0.030,Y -556.060,Z 1083.755,A 0.000,B 0.000,C 90.000,E1 171.894} C_DIS
LIN {X 0.028,Y -562.848,Z 1083.747,A 0.000,B 0.000,C 90.000,E1 170.500} C_DIS
LIN {X 0.210,Y -569.505,Z 1083.740,A 0.000,B 0.000,C 90.000,E1 169.106} C_DIS
LIN {X 0.054,Y -575.818,Z 1083.732,A 0.000,B 0.000,C 90.000,E1 167.757} C_DIS
LIN {X -0.219,Y -580.670,Z 1083.726,A 0.000,B 0.000,C 90.000,E1 166.700} C_DIS
LIN {X 0.128,Y -585.356,Z 1083.720,A 0.000,B 0.000,C 90.000,E1 165.589} C_DIS
LIN {X 0.188,Y -587.672,Z 1083.717,A 0.000,B 0.000,C 90.000,E1 165.046} C_DIS
LIN {X -0.099,Y -593.061,Z 1083.710,A 0.000,B 0.000,C 90.000,E1 163.740} C_DIS
LIN {X -0.009,Y -597.021,Z 1083.704,A 0.000,B 0.000,C 90.000,E1 162.670} C_DIS
LIN {X 0.036,Y -599.880,Z 1083.699,A 0.000,B 0.000,C 90.000,E1 161.873} C_DIS
LIN {X -0.361,Y -603.519,Z 1083.693,A 0.000,B 0.000,C 90.000,E1 160.859} C_DIS
LIN {X 0.259,Y -606.910,Z 1083.688,A 0.000,B 0.000,C 90.000,E1 159.752} C_DIS
LIN {X 0.095,Y -610.917,Z 1083.680,A 0.000,B 0.000,C 90.000,E1 158.465} C_DIS
LIN {X -0.008,Y -614.691,Z 1083.673,A 0.000,B 0.000,C 90.000,E1 157.177} C_DIS
LIN {X 0.181,Y -618.292,Z 1083.666,A 0.000,B 0.000,C 90.000,E1 155.869} C_DIS
LIN {X 0.126,Y -622.276,Z 1083.657,A 0.000,B 0.000,C 90.000,E1 154.332} C_DIS
LIN {X -0.131,Y -625.481,Z 1083.650,A 0.000,B 0.000,C 90.000,E1 153.076} C_DIS
LIN {X 0.249,Y -629.170,Z 1083.642,A 0.000,B 0.000,C 90.000,E1 151.513} C_DIS
LIN {X 0.129,Y -632.022,Z 1083.635,A 0.000,B 0.000,C 90.000,E1 150.255} C_DIS
LIN {X 0.091,Y -635.323,Z 1083.626,A 0.000,B 0.000,C 90.000,E1 148.742} C_DIS
LIN {X -0.137,Y -637.993,Z 1083.619,A 0.000,B 0.000,C 90.000,E1 147.502} C_DIS
LIN {X 0.223,Y -640.531,Z 1083.612,A 0.000,B 0.000,C 90.000,E1 146.215} C_DIS
LIN {X 0.084,Y -642.989,Z 1083.605,A 0.000,B 0.000,C 90.000,E1 144.975} C_DIS
LIN {X 0.353,Y -645.407,Z 1083.599,A 0.000,B 0.000,C 90.000,E1 143.703} C_DIS
LIN {X 0.146,Y -647.741,Z 1083.592,A 0.000,B 0.000,C 90.000,E1 142.477} C_DIS
LIN {X -0.096,Y -650.615,Z 1083.583,A 0.000,B 0.000,C 90.000,E1 141.009} C_DIS
LIN {X -0.287,Y -653.594,Z 1083.575,A 0.000,B 0.000,C 90.000,E1 139.542} C_DIS
LIN {X -0.047,Y -657.084,Z 1083.566,A 0.000,B 0.000,C 90.000,E1 137.796} C_DIS
LIN {X 0.213,Y -661.217,Z 1083.555,A 0.000,B 0.000,C 90.000,E1 135.810} C_DIS
LIN {X 0.125,Y -665.260,Z 1083.545,A 0.000,B 0.000,C 90.000,E1 134.109} C_DIS
LIN {X -0.340,Y -669.558,Z 1083.536,A 0.000,B 0.000,C 90.000,E1 132.447} C_DIS
LIN {X 0.300,Y -674.480,Z 1083.525,A 0.000,B 0.000,C 90.000,E1 130.458} C_DIS
LIN {X 0.057,Y -678.110,Z 1083.517,A 0.000,B 0.000,C 90.000,E1 129.036} C_DIS
LIN {X -0.375,Y -683.081,Z 1083.506,A 0.000,B 0.000,C 90.000,E1 127.156} C_DIS
LIN {X 0.033,Y -686.161,Z 1083.500,A 0.000,B 0.000,C 90.000,E1 125.931} C_DIS
LIN {X -0.283,Y -689.612,Z 1083.492,A 0.000,B 0.000,C 90.000,E1 124.532} C_DIS
LIN {X 0.264,Y -693.652,Z 1083.483,A 0.000,B 0.000,C 90.000,E1 122.832} C_DIS
LIN {X -0.294,Y -697.039,Z 1083.475,A 0.000,B 0.000,C 90.000,E1 121.465} C_DIS
LIN {X -0.125,Y -699.094,Z 1083.469,A 0.000,B 0.000,C 90.000,E1 120.512} C_DIS
LIN {X 0.320,Y -700.774,Z 1083.464,A 0.000,B 0.000,C 90.000,E1 119.539} C_DIS
LIN {X -0.092,Y -701.678,Z 1083.460,A 0.000,B 0.000,C 90.000,E1 118.871} C_DIS
LIN {X 0.391,Y -702.675,Z 1083.455,A 0.000,B 0.000,C 90.000,E1 117.897} C_DIS
LIN {X 0.227,Y -703.752,Z 1083.449,A 0.000,B 0.000,C 90.000,E1 116.744} C_DIS
LIN {X 0.078,Y -704.790,Z 1083.442,A 0.000,B 0.000,C 90.000,E1 115.591} C_DIS
LIN {X -0.285,Y -705.115,Z 1083.440,A 0.000,B 0.000,C 90.000,E1 115.155} C_DIS
LIN {X 0.291,Y -705.169,Z 1083.437,A 0.000,B 0.000,C 90.000,E1 114.643} C_DIS
LIN {X -0.067,Y -704.726,Z 1083.434,A 0.000,B 0.000,C 90.000,E1 114.207} C_DIS
LIN {X 0.218,Y -704.396,Z 1083.433,A 0.000,B 0.000,C 90.000,E1 113.951} C_DIS
LIN {X -0.143,Y -702.787,Z 1083.431,A 0.000,B 0.000,C 90.000,E1 113.515} C_DIS
LIN {X 0.136,Y -701.708,Z 1083.429,A 0.000,B 0.000,C 90.000,E1 113.259} C_DIS
LIN {X -0.242,Y -698.073,Z 1083.427,A 0.000,B 0.000,C 90.000,E1 112.823} C_DIS
LIN {X -0.113,Y -696.951,Z 1083.426,A 0.000,B 0.000,C 90.000,E1 112.695} C_DIS
LIN {X -0.250,Y -695.234,Z 1083.425,A 0.000,B 0.000,C 90.000,E1 112.589} C_DIS
LIN {X 0.332,Y -687.618,Z 1083.424,A 0.000,B 0.000,C 90.000,E1 112.206} C_DIS
LIN {X 0.111,Y -685.664,Z 1083.423,A 0.000,B 0.000,C 90.000,E1 112.153} C_DIS
LIN {X -0.316,Y -684.023,Z 1083.423,A 0.000,B 0.000,C 90.000,E1 112.153} C_DIS
LIN {X -0.049,Y -676.008,Z 1083.422,A 0.000,B 0.000,C 90.000,E1 112.025} C_DIS
LIN {X -0.092,Y -605.458,Z 1083.422,A 0.000,B 0.000,C 90.000,E1 112.025} C_DIS
LIN {X -0.036,Y -601.654,Z 1083.421,A 0.000,B 0.000,C 90.000,E1 111.844} C_DIS
LIN {X 0.167,Y -596.350,Z 1083.419,A 0.000,B 0.000,C 90.000,E1 111.482} C_DIS
LIN {X 0.141,Y -586.221,Z 1083.415,A 0.000,B 0.000,C 90.000,E1 110.663} C_DIS
LIN {X 0.214,Y -579.258,Z 1083.412,A 0.000,B 0.000,C 90.000,E1 110.066} C_DIS
LIN {X -0.209,Y -575.034,Z 1083.410,A 0.000,B 0.000,C 90.000,E1 109.758} C_DIS
LIN {X 0.131,Y -568.948,Z 1083.407,A 0.000,B 0.000,C 90.000,E1 109.268} C_DIS
LIN {X -0.112,Y -560.651,Z 1083.404,A 0.000,B 0.000,C 90.000,E1 108.779} C_DIS
LIN {X -0.154,Y -554.235,Z 1083.402,A 0.000,B 0.000,C 90.000,E1 108.417} C_DIS
LIN {X -0.026,Y -549.251,Z 1083.400,A 0.000,B 0.000,C 90.000,E1 108.055} C_DIS
LIN {X -0.011,Y -547.866,Z 1083.399,A 0.000,B 0.000,C 90.000,E1 107.873} C_DIS
LIN {X -0.053,Y -547.837,Z 1083.399,A 0.000,B 0.000,C 90.000,E1 107.873} C_DIS
LIN {X -0.235,Y -547.527,Z 1083.398,A 0.000,B 0.000,C 90.000,E1 107.638} C_DIS
LIN {X -0.335,Y -547.830,Z 1083.393,A 0.000,B 0.000,C 90.000,E1 106.804} C_DIS
LIN {X -0.184,Y -548.611,Z 1083.387,A 0.000,B 0.000,C 90.000,E1 105.662} C_DIS
LIN {X 0.275,Y -550.013,Z 1083.376,A 0.000,B 0.000,C 90.000,E1 103.647} C_DIS
LIN {X -0.018,Y -551.633,Z 1083.365,A 0.000,B 0.000,C 90.000,E1 101.715} C_DIS
LIN {X 0.029,Y -552.995,Z 1083.357,A 0.000,B 0.000,C 90.000,E1 100.310} C_DIS
LIN {X 0.165,Y -555.131,Z 1083.346,A 0.000,B 0.000,C 90.000,E1 98.341} C_DIS
LIN {X 0.229,Y -556.965,Z 1083.337,A 0.000,B 0.000,C 90.000,E1 96.663} C_DIS
LIN {X 0.062,Y -558.181,Z 1083.331,A 0.000,B 0.000,C 90.000,E1 95.568} C_DIS
LIN {X -0.008,Y -559.369,Z 1083.323,A 0.000,B 0.000,C 90.000,E1 94.188} C_DIS
LIN {X -0.155,Y -560.098,Z 1083.317,A 0.000,B 0.000,C 90.000,E1 93.094} C_DIS
LIN {X -0.145,Y -561.069,Z 1083.308,A 0.000,B 0.000,C 90.000,E1 91.432} C_DIS
LIN {X -0.124,Y -561.775,Z 1083.299,A 0.000,B 0.000,C 90.000,E1 89.771} C_DIS
LIN {X -0.189,Y -562.352,Z 1083.291,A 0.000,B 0.000,C 90.000,E1 88.396} C_DIS
LIN {X -0.233,Y -562.926,Z 1083.283,A 0.000,B 0.000,C 90.000,E1 87.020} C_DIS
LIN {X -0.232,Y -563.459,Z 1083.276,A 0.000,B 0.000,C 90.000,E1 85.641} C_DIS
LIN {X -0.067,Y -564.017,Z 1083.266,A 0.000,B 0.000,C 90.000,E1 83.970} C_DIS
LIN {X -0.049,Y -564.446,Z 1083.259,A 0.000,B 0.000,C 90.000,E1 82.591} C_DIS
LIN {X 0.196,Y -564.997,Z 1083.250,A 0.000,B 0.000,C 90.000,E1 80.914} C_DIS
LIN {X 0.150,Y -565.799,Z 1083.239,A 0.000,B 0.000,C 90.000,E1 78.993} C_DIS
LIN {X 0.236,Y -566.671,Z 1083.228,A 0.000,B 0.000,C 90.000,E1 77.061} C_DIS
LIN {X 0.240,Y -567.953,Z 1083.216,A 0.000,B 0.000,C 90.000,E1 74.866} C_DIS
LIN {X -0.262,Y -569.591,Z 1083.204,A 0.000,B 0.000,C 90.000,E1 72.725} C_DIS
LIN {X -0.010,Y -571.120,Z 1083.193,A 0.000,B 0.000,C 90.000,E1 70.786} C_DIS
LIN {X 0.298,Y -572.286,Z 1083.186,A 0.000,B 0.000,C 90.000,E1 69.390} C_DIS
LIN {X 0.080,Y -573.400,Z 1083.178,A 0.000,B 0.000,C 90.000,E1 68.050} C_DIS
LIN {X 0.313,Y -574.559,Z 1083.171,A 0.000,B 0.000,C 90.000,E1 66.666} C_DIS
LIN {X 0.185,Y -575.782,Z 1083.161,A 0.000,B 0.000,C 90.000,E1 65.049} C_DIS
LIN {X 0.047,Y -576.813,Z 1083.152,A 0.000,B 0.000,C 90.000,E1 63.435} C_DIS
LIN {X -0.053,Y -577.833,Z 1083.143,A 0.000,B 0.000,C 90.000,E1 61.820} C_DIS
LIN {X -0.145,Y -578.792,Z 1083.134,A 0.000,B 0.000,C 90.000,E1 60.205} C_DIS
LIN {X -0.295,Y -579.788,Z 1083.124,A 0.000,B 0.000,C 90.000,E1 58.329} C_DIS
LIN {X -0.273,Y -580.549,Z 1083.115,A 0.000,B 0.000,C 90.000,E1 56.707} C_DIS
LIN {X 0.238,Y -581.131,Z 1083.107,A 0.000,B 0.000,C 90.000,E1 55.308} C_DIS
LIN {X -0.056,Y -581.469,Z 1083.103,A 0.000,B 0.000,C 90.000,E1 54.529} C_DIS
LIN {X 0.007,Y -581.883,Z 1083.095,A 0.000,B 0.000,C 90.000,E1 53.176} C_DIS
LIN {X 0.072,Y -582.125,Z 1083.088,A 0.000,B 0.000,C 90.000,E1 51.823} C_DIS
LIN {X 0.317,Y -582.035,Z 1083.082,A 0.000,B 0.000,C 90.000,E1 50.723} C_DIS
LIN {X 0.282,Y -581.731,Z 1083.075,A 0.000,B 0.000,C 90.000,E1 49.380} C_DIS
LIN {X 0.071,Y -581.348,Z 1083.069,A 0.000,B 0.000,C 90.000,E1 48.324} C_DIS
LIN {X 0.126,Y -580.643,Z 1083.060,A 0.000,B 0.000,C 90.000,E1 46.701} C_DIS
LIN {X -0.135,Y -579.969,Z 1083.054,A 0.000,B 0.000,C 90.000,E1 45.648} C_DIS
LIN {X -0.127,Y -579.325,Z 1083.049,A 0.000,B 0.000,C 90.000,E1 44.838} C_DIS
LIN {X -0.127,Y -578.536,Z 1083.045,A 0.000,B 0.000,C 90.000,E1 44.028} C_DIS
LIN {X -0.140,Y -577.595,Z 1083.040,A 0.000,B 0.000,C 90.000,E1 43.218} C_DIS
LIN {X 0.257,Y -576.557,Z 1083.036,A 0.000,B 0.000,C 90.000,E1 42.366} C_DIS
LIN {X -0.028,Y -575.023,Z 1083.030,A 0.000,B 0.000,C 90.000,E1 41.310} C_DIS
LIN {X 0.042,Y -573.112,Z 1083.023,A 0.000,B 0.000,C 90.000,E1 40.216} C_DIS
LIN {X 0.147,Y -570.966,Z 1083.017,A 0.000,B 0.000,C 90.000,E1 39.116} C_DIS
LIN {X 0.224,Y -568.474,Z 1083.011,A 0.000,B 0.000,C 90.000,E1 38.016} C_DIS
LIN {X 0.350,Y -567.826,Z 1083.010,A 0.000,B 0.000,C 90.000,E1 37.729} C_DIS
LIN {X 0.037,Y -564.603,Z 1083.004,A 0.000,B 0.000,C 90.000,E1 36.664} C_DIS
LIN {X 0.260,Y -562.863,Z 1083.001,A 0.000,B 0.000,C 90.000,E1 36.091} C_DIS
LIN {X -0.088,Y -561.956,Z 1082.999,A 0.000,B 0.000,C 90.000,E1 35.851} C_DIS
LIN {X -0.119,Y -558.717,Z 1082.995,A 0.000,B 0.000,C 90.000,E1 35.025} C_DIS
LIN {X -0.176,Y -555.273,Z 1082.990,A 0.000,B 0.000,C 90.000,E1 34.199} C_DIS
LIN {X -0.270,Y -551.518,Z 1082.985,A 0.000,B 0.000,C 90.000,E1 33.372} C_DIS
LIN {X 0.053,Y -547.299,Z 1082.981,A 0.000,B 0.000,C 90.000,E1 32.498} C_DIS
LIN {X -0.263,Y -542.140,Z 1082.975,A 0.000,B 0.000,C 90.000,E1 31.544} C_DIS
LIN {X 0.092,Y -538.129,Z 1082.971,A 0.000,B 0.000,C 90.000,E1 30.797} C_DIS
LIN {X 0.114,Y -532.126,Z 1082.966,A 0.000,B 0.000,C 90.000,E1 29.795} C_DIS
LIN {X 0.101,Y -527.267,Z 1082.962,A 0.000,B 0.000,C 90.000,E1 29.077} C_DIS
LIN {X -0.103,Y -524.205,Z 1082.959,A 0.000,B 0.000,C 90.000,E1 28.665} C_DIS
LIN {X -0.273,Y -519.808,Z 1082.956,A 0.000,B 0.000,C 90.000,E1 28.103} C_DIS
